    movel([0.183357, -1.188644, -2.683075, -0.840670, 1.570796, 1.754154],accel_mss,speed_ms,0,blend_radius_m)
    movel([0.183318, -1.188232, -2.683266, -0.840892, 1.570796, 1.754114],accel_mss,speed_ms,0,blend_radius_m)
    movel([0.183016, -1.187801, -2.683465, -0.841123, 1.570796, 1.753812],accel_mss,speed_ms,0,blend_radius_m)
    movel([0.182567, -1.187331, -2.683682, -0.841376, 1.570796, 1.753364],accel_mss,speed_ms,0,blend_radius_m)
    movel([0.183152, -1.186492, -2.684069, -0.841828, 1.570796, 1.753948],accel_mss,speed_ms,0,blend_radius_m)
    movel([0.183941, -1.185475, -2.684537, -0.842376, 1.570796, 1.754737],accel_mss,speed_ms,0,blend_radius_m)
    movel([0.184909, -1.184431, -2.685017, -0.842941, 1.570796, 1.755705],accel_mss,speed_ms,0,blend_radius_m)
    movel([0.185946, -1.183470, -2.685457, -0.843461, 1.570796, 1.756743],accel_mss,speed_ms,0,blend_radius_m)
    movel([0.186948, -1.182701, -2.685809, -0.843879, 1.570796, 1.757744],accel_mss,speed_ms,0,blend_radius_m)
    movel([0.187725, -1.182215, -2.686031, -0.844143, 1.570796, 1.758522],accel_mss,speed_ms,0,blend_radius_m)
    movel([0.189510, -1.181449, -2.686380, -0.844559, 1.570796, 1.760306],accel_mss,speed_ms,0,blend_radius_m)
    movel([0.191283, -1.180865, -2.686647, -0.844878, 1.570796, 1.762079],accel_mss,speed_ms,0,blend_radius_m)
    movel([0.194335, -1.179783, -2.687138, -0.845468, 1.570796, 1.765131],accel_mss,speed_ms,0,blend_radius_m)
    movel([0.194860, -1.179431, -2.687298, -0.845660, 1.570796, 1.765656],accel_mss,speed_ms,0,blend_radius_m)
    movel([0.195107, -1.179039, -2.687476, -0.845874, 1.570796, 1.765903],accel_mss,speed_ms,0,blend_radius_m)
    movel([0.194973, -1.178763, -2.687601, -0.846025, 1.570796, 1.765769],accel_mss,speed_ms,0,blend_radius_m)
    movel([0.194450, -1.178756, -2.687604, -0.846029, 1.570796, 1.765246],accel_mss,speed_ms,0,blend_radius_m)
    movel([0.193355, -1.179040, -2.687475, -0.845874, 1.570796, 1.764151],accel_mss,speed_ms,0,blend_radius_m)
    movel([0.188730, -1.180627, -2.686755, -0.845007, 1.570796, 1.759526],accel_mss,speed_ms,0,blend_radius_m)
    movel([0.187737, -1.181042, -2.686566, -0.844781, 1.570796, 1.758533],accel_mss,speed_ms,0,blend_radius_m)
    movel([0.185925, -1.182231, -2.686024, -0.844134, 1.570796, 1.756721],accel_mss,speed_ms,0,blend_radius_m)
    movel([0.184712, -1.183244, -2.685561, -0.843584, 1.570796, 1.755509],accel_mss,speed_ms,0,blend_radius_m)
    movel([0.183607, -1.184345, -2.685056, -0.842987, 1.570796, 1.754403],accel_mss,speed_ms,0,blend_radius_m)
    movel([0.182652, -1.185493, -2.684529, -0.842367, 1.570796, 1.753449],accel_mss,speed_ms,0,blend_radius_m)
    movel([0.181882, -1.186645, -2.683999, -0.841745, 1.570796, 1.752679],accel_mss,speed_ms,0,blend_radius_m)
    movel([0.181412, -1.187532, -2.683589, -0.841268, 1.570796, 1.752208],accel_mss,speed_ms,0,blend_radius_m)
    movel([0.181236, -1.188120, -2.683317, -0.840952, 1.570796, 1.752032],accel_mss,speed_ms,0,blend_radius_m)
    movel([0.181309, -1.188513, -2.683135, -0.840741, 1.570796, 1.752106],accel_mss,speed_ms,0,blend_radius_m)
    movel([0.182133, -1.189002, -2.682909, -0.840478, 1.570796, 1.752929],accel_mss,speed_ms,0,blend_radius_m)
    movel([0.181364, -1.190142, -2.682379, -0.839868, 1.570796, 1.752161],accel_mss,speed_ms,0,blend_radius_m)
    movel([0.180621, -1.191525, -2.681735, -0.839129, 1.570796, 1.751417],accel_mss,speed_ms,0,blend_radius_m)
    movel([0.180458, -1.192089, -2.681472, -0.838828, 1.570796, 1.751254],accel_mss,speed_ms,0,blend_radius_m)
    movel([0.180578, -1.193029, -2.681033, -0.838328, 1.570796, 1.751374],accel_mss,speed_ms,0,blend_radius_m)
    movel([0.180851, -1.193345, -2.680885, -0.838160, 1.570796, 1.751647],accel_mss,speed_ms,0,blend_radius_m)
    movel([0.181819, -1.193755, -2.680692, -0.837942, 1.570796, 1.752615],accel_mss,speed_ms,0,blend_radius_m)
    movel([0.182308, -1.193800, -2.680671, -0.837918, 1.570796, 1.753104],accel_mss,speed_ms,0,blend_radius_m)
    movel([0.188084, -1.193535, -2.680795, -0.838058, 1.570796, 1.758880],accel_mss,speed_ms,0,blend_radius_m)
    movel([0.188322, -1.193692, -2.680722, -0.837975, 1.570796, 1.759118],accel_mss,speed_ms,0,blend_radius_m)
    movel([0.188151, -1.193926, -2.680612, -0.837851, 1.570796, 1.758948],accel_mss,speed_ms,0,blend_radius_m)
    movel([0.185986, -1.194616, -2.680288, -0.837485, 1.570796, 1.756782],accel_mss,speed_ms,0,blend_radius_m)
    movel([0.179630, -1.197004, -2.679163, -0.836222, 1.570796, 1.750426],accel_mss,speed_ms,0,blend_radius_m)
    movel([0.176831, -1.197828, -2.678774, -0.835788, 1.570796, 1.747627],accel_mss,speed_ms,0,blend_radius_m)
    movel([0.174272, -1.198330, -2.678536, -0.835523, 1.570796, 1.745068],accel_mss,speed_ms,0,blend_radius_m)
    movel([0.172010, -1.198496, -2.678457, -0.835436, 1.570796, 1.742806],accel_mss,speed_ms,0,blend_radius_m)
    movel([0.170796, -1.198363, -2.678520, -0.835506, 1.570796, 1.741592],accel_mss,speed_ms,0,blend_radius_m)
    movel([0.170175, -1.197936, -2.678722, -0.835731, 1.570796, 1.740972],accel_mss,speed_ms,0,blend_radius_m)
    movel([0.170106, -1.197645, -2.678860, -0.835884, 1.570796, 1.740903],accel_mss,speed_ms,0,blend_radius_m)
    movel([0.170192, -1.197281, -2.679032, -0.836076, 1.570796, 1.740989],accel_mss,speed_ms,0,blend_radius_m)
    movel([0.171081, -1.196153, -2.679565, -0.836671, 1.570796, 1.741877],accel_mss,speed_ms,0,blend_radius_m)
    movel([0.171201, -1.195957, -2.679657, -0.836775, 1.570796, 1.741997],accel_mss,speed_ms,0,blend_radius_m)
    movel([0.171099, -1.195476, -2.679884, -0.837029, 1.570796, 1.741896],accel_mss,speed_ms,0,blend_radius_m)
    movel([0.170976, -1.195295, -2.679969, -0.837125, 1.570796, 1.741772],accel_mss,speed_ms,0,blend_radius_m)
    movel([0.170326, -1.195000, -2.680108, -0.837281, 1.570796, 1.741123],accel_mss,speed_ms,0,blend_radius_m)
    movel([0.169806, -1.194777, -2.680213, -0.837399, 1.570796, 1.740602],accel_mss,speed_ms,0,blend_radius_m)
    movel([0.169725, -1.194532, -2.680327, -0.837529, 1.570796, 1.740521],accel_mss,speed_ms,0,blend_radius_m)
    movel([0.169784, -1.194220, -2.680474, -0.837695, 1.570796, 1.740581],accel_mss,speed_ms,0,blend_radius_m)
    movel([0.170346, -1.193265, -2.680922, -0.838202, 1.570796, 1.741143],accel_mss,speed_ms,0,blend_radius_m)
    movel([0.171551, -1.191871, -2.681574, -0.838944, 1.570796, 1.742347],accel_mss,speed_ms,0,blend_radius_m)
    movel([0.173401, -1.190152, -2.682375, -0.839862, 1.570796, 1.744197],accel_mss,speed_ms,0,blend_radius_m)
    movel([0.175623, -1.188559, -2.683114, -0.840716, 1.570796, 1.746419],accel_mss,speed_ms,0,blend_radius_m)
    movel([0.177833, -1.187338, -2.683679, -0.841372, 1.570796, 1.748630],accel_mss,speed_ms,0,blend_radius_m)
    movel([0.178746, -1.186974, -2.683847, -0.841568, 1.570796, 1.749542],accel_mss,speed_ms,0,blend_radius_m)
    movel([0.180052, -1.186660, -2.683992, -0.841737, 1.570796, 1.750848],accel_mss,speed_ms,0,blend_radius_m)
    movel([0.180327, -1.186549, -2.684043, -0.841797, 1.570796, 1.751123],accel_mss,speed_ms,0,blend_radius_m)
    movel([0.180720, -1.186157, -2.684224, -0.842008, 1.570796, 1.751516],accel_mss,speed_ms,0,blend_radius_m)
    movel([0.180901, -1.185757, -2.684408, -0.842224, 1.570796, 1.751698],accel_mss,speed_ms,0,blend_radius_m)
    movel([0.180851, -1.185515, -2.684519, -0.842355, 1.570796, 1.751647],accel_mss,speed_ms,0,blend_radius_m)
    movel([0.180544, -1.185423, -2.684562, -0.842405, 1.570796, 1.751341],accel_mss,speed_ms,0,blend_radius_m)
    movel([0.179921, -1.185486, -2.684533, -0.842371, 1.570796, 1.750718],accel_mss,speed_ms,0,blend_radius_m)
    movel([0.178586, -1.185838, -2.684371, -0.842181, 1.570796, 1.749382],accel_mss,speed_ms,0,blend_radius_m)
    movel([0.177208, -1.186449, -2.684089, -0.841851, 1.570796, 1.748004],accel_mss,speed_ms,0,blend_radius_m)
    movel([0.175555, -1.187413, -2.683644, -0.841332, 1.570796, 1.746352],accel_mss,speed_ms,0,blend_radius_m)
    movel([0.173939, -1.188522, -2.683131, -0.840736, 1.570796, 1.744736],accel_mss,speed_ms,0,blend_radius_m)
    movel([0.172391, -1.189757, -2.682558, -0.840074, 1.570796, 1.743187],accel_mss,speed_ms,0,blend_radius_m)
    movel([0.170920, -1.191108, -2.681930, -0.839352, 1.570796, 1.741716],accel_mss,speed_ms,0,blend_radius_m)
    movel([0.169840, -1.192310, -2.681369, -0.838710, 1.570796, 1.740637],accel_mss,speed_ms,0,blend_radius_m)
    movel([0.168953, -1.193603, -2.680764, -0.838022, 1.570796, 1.739749],accel_mss,speed_ms,0,blend_radius_m)
    movel([0.168565, -1.194208, -2.680480, -0.837701, 1.570796, 1.739361],accel_mss,speed_ms,0,blend_radius_m)
    movel([0.167841, -1.194873, -2.680167, -0.837348, 1.570796, 1.738638],accel_mss,speed_ms,0,blend_radius_m)
    movel([0.167132, -1.195268, -2.679981, -0.837139, 1.570796, 1.737928],accel_mss,speed_ms,0,blend_radius_m)
    movel([0.164862, -1.196685, -2.679314, -0.836390, 1.570796, 1.735658],accel_mss,speed_ms,0,blend_radius_m)
    movel([0.162528, -1.198602, -2.678407, -0.835380, 1.570796, 1.733324],accel_mss,speed_ms,0,blend_radius_m)
    movel([0.160445, -1.200728, -2.677396, -0.834265, 1.570796, 1.731242],accel_mss,speed_ms,0,blend_radius_m)
    movel([0.159641, -1.201726, -2.676920, -0.833743, 1.570796, 1.730437],accel_mss,speed_ms,0,blend_radius_m)
    movel([0.158201, -1.203864, -2.675896, -0.832628, 1.570796, 1.728998],accel_mss,speed_ms,0,blend_radius_m)
    movel([0.158043, -1.203914, -2.675872, -0.832602, 1.570796, 1.728839],accel_mss,speed_ms,0,blend_radius_m)
    movel([0.157841, -1.203774, -2.675940, -0.832675, 1.570796, 1.728637],accel_mss,speed_ms,0,blend_radius_m)
    movel([0.157600, -1.203660, -2.675994, -0.832735, 1.570796, 1.728397],accel_mss,speed_ms,0,blend_radius_m)
    movel([0.157314, -1.203744, -2.675954, -0.832691, 1.570796, 1.728111],accel_mss,speed_ms,0,blend_radius_m)
    movel([0.156829, -1.204106, -2.675780, -0.832503, 1.570796, 1.727625],accel_mss,speed_ms,0,blend_radius_m)
    movel([0.153276, -1.207330, -2.674226, -0.830833, 1.570796, 1.724072],accel_mss,speed_ms,0,blend_radius_m)
    movel([0.151027, -1.209704, -2.673074, -0.829610, 1.570796, 1.721823],accel_mss,speed_ms,0,blend_radius_m)
    movel([0.148903, -1.212185, -2.671864, -0.828340, 1.570796, 1.719700],accel_mss,speed_ms,0,blend_radius_m)
    movel([0.147125, -1.214534, -2.670712, -0.827143, 1.570796, 1.717921],accel_mss,speed_ms,0,blend_radius_m)
    movel([0.146009, -1.216173, -2.669904, -0.826312, 1.570796, 1.716805],accel_mss,speed_ms,0,blend_radius_m)
    movel([0.145534, -1.217059, -2.669466, -0.825864, 1.570796, 1.716330],accel_mss,speed_ms,0,blend_radius_m)
    movel([0.145529, -1.217471, -2.669262, -0.825656, 1.570796, 1.716326],accel_mss,speed_ms,0,blend_radius_m)
    movel([0.145867, -1.217578, -2.669209, -0.825602, 1.570796, 1.716664],accel_mss,speed_ms,0,blend_radius_m)
    movel([0.146124, -1.217471, -2.669262, -0.825656, 1.570796, 1.716921],accel_mss,speed_ms,0,blend_radius_m)
    movel([0.146381, -1.217258, -2.669368, -0.825763, 1.570796, 1.717177],accel_mss,speed_ms,0,blend_radius_m)
    movel([0.148924, -1.213700, -2.671122, -0.827568, 1.570796, 1.719721],accel_mss,speed_ms,0,blend_radius_m)
    movel([0.151184, -1.210948, -2.672468, -0.828972, 1.570796, 1.721980],accel_mss,speed_ms,0,blend_radius_m)
    movel([0.153647, -1.208297, -2.673758, -0.830334, 1.570796, 1.724443],accel_mss,speed_ms,0,blend_radius_m)
    movel([0.156117, -1.205971, -2.674882, -0.831535, 1.570796, 1.726914],accel_mss,speed_ms,0,blend_radius_m)
    movel([0.157615, -1.204719, -2.675486, -0.832184, 1.570796, 1.728411],accel_mss,speed_ms,0,blend_radius_m)
    movel([0.157396, -1.205607, -2.675058, -0.831724, 1.570796, 1.728192],accel_mss,speed_ms,0,blend_radius_m)
    movel([0.157289, -1.205968, -2.674884, -0.831537, 1.570796, 1.728085],accel_mss,speed_ms,0,blend_radius_m)
    movel([0.157248, -1.206792, -2.674486, -0.831110, 1.570796, 1.728045],accel_mss,speed_ms,0,blend_radius_m)
    movel([0.157510, -1.207083, -2.674346, -0.830960, 1.570796, 1.728307],accel_mss,speed_ms,0,blend_radius_m)
    movel([0.158082, -1.207177, -2.674300, -0.830912, 1.570796, 1.728878],accel_mss,speed_ms,0,blend_radius_m)
    movel([0.159104, -1.207089, -2.674343, -0.830957, 1.570796, 1.729901],accel_mss,speed_ms,0,blend_radius_m)
    movel([0.161055, -1.206656, -2.674552, -0.831181, 1.570796, 1.731852],accel_mss,speed_ms,0,blend_radius_m)
    movel([0.161633, -1.206359, -2.674695, -0.831334, 1.570796, 1.732429],accel_mss,speed_ms,0,blend_radius_m)
    movel([0.161996, -1.205991, -2.674873, -0.831525, 1.570796, 1.732793],accel_mss,speed_ms,0,blend_radius_m)
    movel([0.162127, -1.205617, -2.675053, -0.831718, 1.570796, 1.732924],accel_mss,speed_ms,0,blend_radius_m)
    movel([0.161992, -1.205417, -2.675150, -0.831822, 1.570796, 1.732788],accel_mss,speed_ms,0,blend_radius_m)
    movel([0.161506, -1.205409, -2.675154, -0.831826, 1.570796, 1.732303],accel_mss,speed_ms,0,blend_radius_m)
    movel([0.159027, -1.205918, -2.674908, -0.831563, 1.570796, 1.729824],accel_mss,speed_ms,0,blend_radius_m)
    movel([0.158633, -1.205765, -2.674982, -0.831642, 1.570796, 1.729429],accel_mss,speed_ms,0,blend_radius_m)
    movel([0.158690, -1.205254, -2.675228, -0.831907, 1.570796, 1.729487],accel_mss,speed_ms,0,blend_radius_m)
    movel([0.159555, -1.203686, -2.675982, -0.832721, 1.570796, 1.730351],accel_mss,speed_ms,0,blend_radius_m)
    movel([0.161064, -1.201525, -2.677016, -0.833848, 1.570796, 1.731861],accel_mss,speed_ms,0,blend_radius_m)
    movel([0.163073, -1.199370, -2.678042, -0.834977, 1.570796, 1.733869],accel_mss,speed_ms,0,blend_radius_m)
    movel([0.165272, -1.197525, -2.678917, -0.835947, 1.570796, 1.736068],accel_mss,speed_ms,0,blend_radius_m)
    movel([0.166291, -1.196848, -2.679237, -0.836304, 1.570796, 1.737087],accel_mss,speed_ms,0,blend_radius_m)
    movel([0.167890, -1.196069, -2.679604, -0.836715, 1.570796, 1.738686],accel_mss,speed_ms,0,blend_radius_m)
    movel([0.168251, -1.195979, -2.679647, -0.836763, 1.570796, 1.739048],accel_mss,speed_ms,0,blend_radius_m)
    movel([0.168882, -1.196151, -2.679566, -0.836672, 1.570796, 1.739679],accel_mss,speed_ms,0,blend_radius_m)
    movel([0.169124, -1.196310, -2.679491, -0.836588, 1.570796, 1.739920],accel_mss,speed_ms,0,blend_radius_m)
    movel([0.169263, -1.196631, -2.679339, -0.836418, 1.570796, 1.740059],accel_mss,speed_ms,0,blend_radius_m)
    movel([0.169187, -1.196810, -2.679255, -0.836324, 1.570796, 1.739984],accel_mss,speed_ms,0,blend_radius_m)
    movel([0.168789, -1.197977, -2.678703, -0.835709, 1.570796, 1.739586],accel_mss,speed_ms,0,blend_radius_m)
    movel([0.168749, -1.198411, -2.678497, -0.835481, 1.570796, 1.739546],accel_mss,speed_ms,0,blend_radius_m)
    movel([0.168985, -1.199003, -2.678217, -0.835170, 1.570796, 1.739781],accel_mss,speed_ms,0,blend_radius_m)
    movel([0.169337, -1.199309, -2.678071, -0.835009, 1.570796, 1.740134],accel_mss,speed_ms,0,blend_radius_m)
    movel([0.170273, -1.199713, -2.677879, -0.834797, 1.570796, 1.741070],accel_mss,speed_ms,0,blend_radius_m)
    movel([0.170932, -1.199776, -2.677850, -0.834764, 1.570796, 1.741729],accel_mss,speed_ms,0,blend_radius_m)
    movel([0.173806, -1.199710, -2.677881, -0.834798, 1.570796, 1.744603],accel_mss,speed_ms,0,blend_radius_m)
    movel([0.169997, -1.201753, -2.676907, -0.833729, 1.570796, 1.740793],accel_mss,speed_ms,0,blend_radius_m)
    movel([0.164056, -1.205160, -2.675273, -0.831955, 1.570796, 1.734852],accel_mss,speed_ms,0,blend_radius_m)
    movel([0.158222, -1.208931, -2.673450, -0.830008, 1.570796, 1.729018],accel_mss,speed_ms,0,blend_radius_m)
    movel([0.155609, -1.210782, -2.672549, -0.829057, 1.570796, 1.726406],accel_mss,speed_ms,0,blend_radius_m)
    movel([0.153043, -1.212728, -2.671598, -0.828063, 1.570796, 1.723839],accel_mss,speed_ms,0,blend_radius_m)
    movel([0.148093, -1.216872, -2.669559, -0.825958, 1.570796, 1.718889],accel_mss,speed_ms,0,blend_radius_m)
    movel([0.145657, -1.219114, -2.668447, -0.824828, 1.570796, 1.716453],accel_mss,speed_ms,0,blend_radius_m)
    movel([0.141026, -1.223786, -2.666112, -0.822491, 1.570796, 1.711822],accel_mss,speed_ms,0,blend_radius_m)
    movel([0.138839, -1.226205, -2.664893, -0.821290, 1.570796, 1.709635],accel_mss,speed_ms,0,blend_radius_m)
    movel([0.134113, -1.231833, -2.662032, -0.818524, 1.570796, 1.704910],accel_mss,speed_ms,0,blend_radius_m)
    movel([0.129720, -1.237546, -2.659090, -0.815754, 1.570796, 1.700516],accel_mss,speed_ms,0,blend_radius_m)
    movel([0.127006, -1.241371, -2.657098, -0.813920, 1.570796, 1.697802],accel_mss,speed_ms,0,blend_radius_m)
    movel([0.124468, -1.245218, -2.655078, -0.812093, 1.570796, 1.695265],accel_mss,speed_ms,0,blend_radius_m)
    movel([0.122226, -1.248912, -2.653121, -0.810355, 1.570796, 1.693023],accel_mss,speed_ms,0,blend_radius_m)
    movel([0.120184, -1.252606, -2.651149, -0.808634, 1.570796, 1.690981],accel_mss,speed_ms,0,blend_radius_m)
    movel([0.118156, -1.256650, -2.648970, -0.806769, 1.570796, 1.688952],accel_mss,speed_ms,0,blend_radius_m)
    movel([0.116335, -1.260667, -2.646787, -0.804935, 1.570796, 1.687131],accel_mss,speed_ms,0,blend_radius_m)
    movel([0.114295, -1.265566, -2.644097, -0.802726, 1.570796, 1.685091],accel_mss,speed_ms,0,blend_radius_m)
    movel([0.112409, -1.270417, -2.641405, -0.800567, 1.570796, 1.683205],accel_mss,speed_ms,0,blend_radius_m)
    movel([0.110443, -1.275872, -2.638343, -0.798175, 1.570796, 1.681240],accel_mss,speed_ms,0,blend_radius_m)
    movel([0.109095, -1.280175, -2.635901, -0.796313, 1.570796, 1.679892],accel_mss,speed_ms,0,blend_radius_m)
    movel([0.108198, -1.283839, -2.633803, -0.794747, 1.570796, 1.678994],accel_mss,speed_ms,0,blend_radius_m)
    movel([0.107629, -1.287288, -2.631813, -0.793288, 1.570796, 1.678425],accel_mss,speed_ms,0,blend_radius_m)
    movel([0.107418, -1.289676, -2.630427, -0.792286, 1.570796, 1.678214],accel_mss,speed_ms,0,blend_radius_m)
    movel([0.107364, -1.291997, -2.629072, -0.791320, 1.570796, 1.678161],accel_mss,speed_ms,0,blend_radius_m)
    movel([0.107481, -1.294116, -2.627829, -0.790444, 1.570796, 1.678278],accel_mss,speed_ms,0,blend_radius_m)
    movel([0.107776, -1.296142, -2.626636, -0.789612, 1.570796, 1.678573],accel_mss,speed_ms,0,blend_radius_m)
    movel([0.108341, -1.298654, -2.625148, -0.788587, 1.570796, 1.679137],accel_mss,speed_ms,0,blend_radius_m)
    movel([0.109047, -1.301076, -2.623707, -0.787607, 1.570796, 1.679843],accel_mss,speed_ms,0,blend_radius_m)
    movel([0.111736, -1.308914, -2.618988, -0.784486, 1.570796, 1.682533],accel_mss,speed_ms,0,blend_radius_m)
    movel([0.113063, -1.312631, -2.616723, -0.783035, 1.570796, 1.683860],accel_mss,speed_ms,0,blend_radius_m)
    movel([0.112154, -1.313491, -2.616196, -0.782702, 1.570796, 1.682950],accel_mss,speed_ms,0,blend_radius_m)
    movel([0.110554, -1.315098, -2.615210, -0.782082, 1.570796, 1.681350],accel_mss,speed_ms,0,blend_radius_m)
    movel([0.105604, -1.320526, -2.611850, -0.780012, 1.570796, 1.676400],accel_mss,speed_ms,0,blend_radius_m)
    movel([0.103992, -1.322440, -2.610657, -0.779292, 1.570796, 1.674788],accel_mss,speed_ms,0,blend_radius_m)
    movel([0.101936, -1.325101, -2.608989, -0.778299, 1.570796, 1.672733],accel_mss,speed_ms,0,blend_radius_m)
    movel([0.100022, -1.327790, -2.607294, -0.777305, 1.570796, 1.670818],accel_mss,speed_ms,0,blend_radius_m)
    movel([0.098207, -1.330560, -2.605538, -0.776291, 1.570796, 1.669003],accel_mss,speed_ms,0,blend_radius_m)
    movel([0.096539, -1.333341, -2.603764, -0.775284, 1.570796, 1.667335],accel_mss,speed_ms,0,blend_radius_m)
    movel([0.095051, -1.336061, -2.602020, -0.774309, 1.570796, 1.665848],accel_mss,speed_ms,0,blend_radius_m)
    movel([0.093714, -1.338778, -2.600266, -0.773345, 1.570796, 1.664510],accel_mss,speed_ms,0,blend_radius_m)
    movel([0.092625, -1.341300, -2.598630, -0.772459, 1.570796, 1.663421],accel_mss,speed_ms,0,blend_radius_m)
    movel([0.091710, -1.343801, -2.596999, -0.771589, 1.570796, 1.662507],accel_mss,speed_ms,0,blend_radius_m)
    movel([0.090931, -1.346349, -2.595328, -0.770712, 1.570796, 1.661727],accel_mss,speed_ms,0,blend_radius_m)
    movel([0.090290, -1.348864, -2.593671, -0.769855, 1.570796, 1.661086],accel_mss,speed_ms,0,blend_radius_m)
    movel([0.089357, -1.353982, -2.590270, -0.768137, 1.570796, 1.660153],accel_mss,speed_ms,0,blend_radius_m)
    movel([0.089065, -1.356593, -2.588520, -0.767275, 1.570796, 1.659861],accel_mss,speed_ms,0,blend_radius_m)
    movel([0.088856, -1.361787, -2.585013, -0.765589, 1.570796, 1.659653],accel_mss,speed_ms,0,blend_radius_m)
    movel([0.088925, -1.364369, -2.583255, -0.764764, 1.570796, 1.659721],accel_mss,speed_ms,0,blend_radius_m)
    movel([0.089318, -1.368741, -2.580258, -0.763390, 1.570796, 1.660114],accel_mss,speed_ms,0,blend_radius_m)
    movel([0.090062, -1.372927, -2.577362, -0.762100, 1.570796, 1.660858],accel_mss,speed_ms,0,blend_radius_m)
    movel([0.091178, -1.377118, -2.574438, -0.760833, 1.570796, 1.661974],accel_mss,speed_ms,0,blend_radius_m)
    movel([0.092594, -1.381119, -2.571623, -0.759647, 1.570796, 1.663390],accel_mss,speed_ms,0,blend_radius_m)
    movel([0.094363, -1.385075, -2.568817, -0.758497, 1.570796, 1.665160],accel_mss,speed_ms,0,blend_radius_m)
    movel([0.096417, -1.388825, -2.566136, -0.757428, 1.570796, 1.667214],accel_mss,speed_ms,0,blend_radius_m)
    movel([0.098800, -1.392482, -2.563503, -0.756405, 1.570796, 1.669596],accel_mss,speed_ms,0,blend_radius_m)
    movel([0.101432, -1.395933, -2.560999, -0.755457, 1.570796, 1.672228],accel_mss,speed_ms,0,blend_radius_m)
    movel([0.103048, -1.397724, -2.559693, -0.754972, 1.570796, 1.673844],accel_mss,speed_ms,0,blend_radius_m)
    movel([0.104830, -1.399364, -2.558493, -0.754532, 1.570796, 1.675626],accel_mss,speed_ms,0,blend_radius_m)
    movel([0.106498, -1.400557, -2.557618, -0.754215, 1.570796, 1.677295],accel_mss,speed_ms,0,blend_radius_m)
    movel([0.108382, -1.401515, -2.556913, -0.753961, 1.570796, 1.679178],accel_mss,speed_ms,0,blend_radius_m)
    movel([0.110318, -1.402168, -2.556432, -0.753789, 1.570796, 1.681114],accel_mss,speed_ms,0,blend_radius_m)
    movel([0.112427, -1.402562, -2.556141, -0.753686, 1.570796, 1.683223],accel_mss,speed_ms,0,blend_radius_m)
    movel([0.114808, -1.402728, -2.556019, -0.753642, 1.570796, 1.685604],accel_mss,speed_ms,0,blend_radius_m)
    movel([0.117295, -1.402659, -2.556070, -0.753660, 1.570796, 1.688091],accel_mss,speed_ms,0,blend_radius_m)
    movel([0.119116, -1.402423, -2.556244, -0.753722, 1.570796, 1.689913],accel_mss,speed_ms,0,blend_radius_m)
    movel([0.121505, -1.401921, -2.556614, -0.753854, 1.570796, 1.692302],accel_mss,speed_ms,0,blend_radius_m)
    movel([0.123903, -1.401300, -2.557071, -0.754018, 1.570796, 1.694699],accel_mss,speed_ms,0,blend_radius_m)
    movel([0.125742, -1.400674, -2.557532, -0.754184, 1.570796, 1.696539],accel_mss,speed_ms,0,blend_radius_m)
    movel([0.129029, -1.399183, -2.558625, -0.754580, 1.570796, 1.699825],accel_mss,speed_ms,0,blend_radius_m)
    movel([0.130586, -1.398328, -2.559251, -0.754809, 1.570796, 1.701382],accel_mss,speed_ms,0,blend_radius_m)
    movel([0.132111, -1.397384, -2.559941, -0.755064, 1.570796, 1.702908],accel_mss,speed_ms,0,blend_radius_m)
    movel([0.133568, -1.396370, -2.560681, -0.755338, 1.570796, 1.704364],accel_mss,speed_ms,0,blend_radius_m)
    movel([0.134973, -1.395280, -2.561474, -0.755635, 1.570796, 1.705769],accel_mss,speed_ms,0,blend_radius_m)
    movel([0.136322, -1.394110, -2.562324, -0.755955, 1.570796, 1.707118],accel_mss,speed_ms,0,blend_radius_m)
    movel([0.137604, -1.392877, -2.563216, -0.756295, 1.570796, 1.708400],accel_mss,speed_ms,0,blend_radius_m)
    movel([0.139420, -1.390830, -2.564695, -0.756864, 1.570796, 1.710217],accel_mss,speed_ms,0,blend_radius_m)
    movel([0.140117, -1.389881, -2.565378, -0.757130, 1.570796, 1.710913],accel_mss,speed_ms,0,blend_radius_m)
    movel([0.140711, -1.388907, -2.566077, -0.757405, 1.570796, 1.711508],accel_mss,speed_ms,0,blend_radius_m)
    movel([0.141155, -1.387998, -2.566729, -0.757662, 1.570796, 1.711951],accel_mss,speed_ms,0,blend_radius_m)
    movel([0.141480, -1.387090, -2.567379, -0.757920, 1.570796, 1.712276],accel_mss,speed_ms,0,blend_radius_m)
    movel([0.141680, -1.386204, -2.568012, -0.758173, 1.570796, 1.712477],accel_mss,speed_ms,0,blend_radius_m)
    movel([0.141752, -1.385350, -2.568621, -0.758418, 1.570796, 1.712549],accel_mss,speed_ms,0,blend_radius_m)
    movel([0.141579, -1.384188, -2.569448, -0.758753, 1.570796, 1.712375],accel_mss,speed_ms,0,blend_radius_m)
    movel([0.141052, -1.383273, -2.570098, -0.759018, 1.570796, 1.711849],accel_mss,speed_ms,0,blend_radius_m)
    movel([0.140042, -1.382449, -2.570682, -0.759258, 1.570796, 1.710838],accel_mss,speed_ms,0,blend_radius_m)
    movel([0.138322, -1.381549, -2.571319, -0.759521, 1.570796, 1.709118],accel_mss,speed_ms,0,blend_radius_m)
    movel([0.135744, -1.380110, -2.572335, -0.759944, 1.570796, 1.706541],accel_mss,speed_ms,0,blend_radius_m)
    movel([0.130444, -1.376520, -2.574857, -0.761012, 1.570796, 1.701240],accel_mss,speed_ms,0,blend_radius_m)
    movel([0.125164, -1.372833, -2.577428, -0.762129, 1.570796, 1.695960],accel_mss,speed_ms,0,blend_radius_m)
    movel([0.122027, -1.370380, -2.579127, -0.762882, 1.570796, 1.692823],accel_mss,speed_ms,0,blend_radius_m)
    movel([0.119338, -1.367897, -2.580839, -0.763653, 1.570796, 1.690134],accel_mss,speed_ms,0,blend_radius_m)
    movel([0.117149, -1.365481, -2.582496, -0.764412, 1.570796, 1.687945],accel_mss,speed_ms,0,blend_radius_m)
    movel([0.115330, -1.362974, -2.584206, -0.765209, 1.570796, 1.686126],accel_mss,speed_ms,0,blend_radius_m)
    movel([0.113763, -1.360220, -2.586075, -0.766094, 1.570796, 1.684560],accel_mss,speed_ms,0,blend_radius_m)
    movel([0.112264, -1.356613, -2.588508, -0.767269, 1.570796, 1.683061],accel_mss,speed_ms,0,blend_radius_m)
    movel([0.111758, -1.354856, -2.589685, -0.767848, 1.570796, 1.682554],accel_mss,speed_ms,0,blend_radius_m)
    movel([0.111393, -1.353018, -2.590913, -0.768458, 1.570796, 1.682190],accel_mss,speed_ms,0,blend_radius_m)
    movel([0.111182, -1.351138, -2.592164, -0.769087, 1.570796, 1.681978],accel_mss,speed_ms,0,blend_radius_m)
    movel([0.111120, -1.349189, -2.593456, -0.769745, 1.570796, 1.681917],accel_mss,speed_ms,0,blend_radius_m)
    movel([0.111200, -1.347063, -2.594858, -0.770467, 1.570796, 1.681997],accel_mss,speed_ms,0,blend_radius_m)
    movel([0.111417, -1.344885, -2.596289, -0.771215, 1.570796, 1.682214],accel_mss,speed_ms,0,blend_radius_m)
    movel([0.112119, -1.340910, -2.598884, -0.772595, 1.570796, 1.682915],accel_mss,speed_ms,0,blend_radius_m)
    movel([0.112599, -1.339021, -2.600109, -0.773259, 1.570796, 1.683395],accel_mss,speed_ms,0,blend_radius_m)
    movel([0.113189, -1.337110, -2.601344, -0.773935, 1.570796, 1.683985],accel_mss,speed_ms,0,blend_radius_m)
    movel([0.114704, -1.333261, -2.603815, -0.775313, 1.570796, 1.685501],accel_mss,speed_ms,0,blend_radius_m)
    movel([0.116745, -1.329144, -2.606437, -0.776808, 1.570796, 1.687541],accel_mss,speed_ms,0,blend_radius_m)
    movel([0.119880, -1.323906, -2.609739, -0.778744, 1.570796, 1.690677],accel_mss,speed_ms,0,blend_radius_m)
    movel([0.120321, -1.323329, -2.610101, -0.778960, 1.570796, 1.691117],accel_mss,speed_ms,0,blend_radius_m)
    movel([0.120558, -1.323269, -2.610138, -0.778982, 1.570796, 1.691354],accel_mss,speed_ms,0,blend_radius_m)
    movel([0.121259, -1.324012, -2.609673, -0.778705, 1.570796, 1.692056],accel_mss,speed_ms,0,blend_radius_m)
    movel([0.124898, -1.328474, -2.606861, -0.777054, 1.570796, 1.695694],accel_mss,speed_ms,0,blend_radius_m)
    movel([0.128998, -1.333445, -2.603698, -0.775246, 1.570796, 1.699794],accel_mss,speed_ms,0,blend_radius_m)
    movel([0.132146, -1.336702, -2.601607, -0.774080, 1.570796, 1.702943],accel_mss,speed_ms,0,blend_radius_m)
    movel([0.135997, -1.339924, -2.599524, -0.772941, 1.570796, 1.706793],accel_mss,speed_ms,0,blend_radius_m)
    movel([0.142877, -1.345098, -2.596150, -0.771141, 1.570796, 1.713674],accel_mss,speed_ms,0,blend_radius_m)
    movel([0.146737, -1.347989, -2.594248, -0.770152, 1.570796, 1.717533],accel_mss,speed_ms,0,blend_radius_m)
    movel([0.145430, -1.350508, -2.592582, -0.769299, 1.570796, 1.716226],accel_mss,speed_ms,0,blend_radius_m)
    movel([0.144148, -1.353044, -2.590896, -0.768449, 1.570796, 1.714944],accel_mss,speed_ms,0,blend_radius_m)
    movel([0.143499, -1.354516, -2.589912, -0.767960, 1.570796, 1.714295],accel_mss,speed_ms,0,blend_radius_m)
    movel([0.143109, -1.355763, -2.589078, -0.767548, 1.570796, 1.713905],accel_mss,speed_ms,0,blend_radius_m)
    movel([0.142789, -1.357342, -2.588017, -0.767030, 1.570796, 1.713585],accel_mss,speed_ms,0,blend_radius_m)
    movel([0.142603, -1.358764, -2.587059, -0.766566, 1.570796, 1.713399],accel_mss,speed_ms,0,blend_radius_m)
    movel([0.142636, -1.359633, -2.586473, -0.766284, 1.570796, 1.713432],accel_mss,speed_ms,0,blend_radius_m)
    movel([0.142888, -1.360224, -2.586073, -0.766092, 1.570796, 1.713684],accel_mss,speed_ms,0,blend_radius_m)
    movel([0.143400, -1.360709, -2.585744, -0.765936, 1.570796, 1.714197],accel_mss,speed_ms,0,blend_radius_m)
    movel([0.144238, -1.360996, -2.585550, -0.765843, 1.570796, 1.715035],accel_mss,speed_ms,0,blend_radius_m)
    movel([0.145422, -1.360988, -2.585555, -0.765846, 1.570796, 1.716218],accel_mss,speed_ms,0,blend_radius_m)
    movel([0.146844, -1.360690, -2.585757, -0.765942, 1.570796, 1.717640],accel_mss,speed_ms,0,blend_radius_m)
    movel([0.148392, -1.360123, -2.586141, -0.766125, 1.570796, 1.719189],accel_mss,speed_ms,0,blend_radius_m)
    movel([0.150333, -1.359097, -2.586834, -0.766457, 1.570796, 1.721129],accel_mss,speed_ms,0,blend_radius_m)
    movel([0.152645, -1.357534, -2.587888, -0.766967, 1.570796, 1.723442],accel_mss,speed_ms,0,blend_radius_m)
    movel([0.154989, -1.355690, -2.589126, -0.767572, 1.570796, 1.725785],accel_mss,speed_ms,0,blend_radius_m)
    movel([0.157035, -1.353806, -2.590387, -0.768196, 1.570796, 1.727831],accel_mss,speed_ms,0,blend_radius_m)
    movel([0.157857, -1.352980, -2.590939, -0.768471, 1.570796, 1.728653],accel_mss,speed_ms,0,blend_radius_m)
    movel([0.160075, -1.353110, -2.590851, -0.768427, 1.570796, 1.730871],accel_mss,speed_ms,0,blend_radius_m)
    movel([0.163680, -1.353196, -2.590794, -0.768399, 1.570796, 1.734476],accel_mss,speed_ms,0,blend_radius_m)
    movel([0.166554, -1.352939, -2.590966, -0.768484, 1.570796, 1.737350],accel_mss,speed_ms,0,blend_radius_m)
    movel([0.167816, -1.352675, -2.591142, -0.768572, 1.570796, 1.738612],accel_mss,speed_ms,0,blend_radius_m)
    movel([0.169098, -1.352297, -2.591393, -0.768699, 1.570796, 1.739894],accel_mss,speed_ms,0,blend_radius_m)
    movel([0.170370, -1.351809, -2.591718, -0.768862, 1.570796, 1.741166],accel_mss,speed_ms,0,blend_radius_m)
    movel([0.171634, -1.351213, -2.592114, -0.769062, 1.570796, 1.742430],accel_mss,speed_ms,0,blend_radius_m)
    movel([0.172833, -1.350504, -2.592584, -0.769300, 1.570796, 1.743629],accel_mss,speed_ms,0,blend_radius_m)
    movel([0.174191, -1.349527, -2.593232, -0.769630, 1.570796, 1.744987],accel_mss,speed_ms,0,blend_radius_m)
    movel([0.175450, -1.348490, -2.593917, -0.769981, 1.570796, 1.746247],accel_mss,speed_ms,0,blend_radius_m)
    movel([0.176314, -1.347609, -2.594499, -0.770281, 1.570796, 1.747111],accel_mss,speed_ms,0,blend_radius_m)
    movel([0.177079, -1.346528, -2.595211, -0.770651, 1.570796, 1.747876],accel_mss,speed_ms,0,blend_radius_m)
    movel([0.177589, -1.345410, -2.595945, -0.771034, 1.570796, 1.748385],accel_mss,speed_ms,0,blend_radius_m)
    movel([0.177789, -1.344366, -2.596630, -0.771394, 1.570796, 1.748585],accel_mss,speed_ms,0,blend_radius_m)
    movel([0.177666, -1.343435, -2.597238, -0.771716, 1.570796, 1.748462],accel_mss,speed_ms,0,blend_radius_m)
    movel([0.177157, -1.342384, -2.597924, -0.772081, 1.570796, 1.747953],accel_mss,speed_ms,0,blend_radius_m)
    movel([0.176397, -1.341524, -2.598484, -0.772381, 1.570796, 1.747193],accel_mss,speed_ms,0,blend_radius_m)
    movel([0.175032, -1.340441, -2.599188, -0.772760, 1.570796, 1.745828],accel_mss,speed_ms,0,blend_radius_m)
    movel([0.171836, -1.338404, -2.600508, -0.773477, 1.570796, 1.742632],accel_mss,speed_ms,0,blend_radius_m)
    movel([0.174790, -1.334338, -2.603126, -0.774925, 1.570796, 1.745587],accel_mss,speed_ms,0,blend_radius_m)
    movel([0.180012, -1.327030, -2.607774, -0.777585, 1.570796, 1.750808],accel_mss,speed_ms,0,blend_radius_m)
    movel([0.182142, -1.323855, -2.609771, -0.778763, 1.570796, 1.752938],accel_mss,speed_ms,0,blend_radius_m)
    movel([0.184172, -1.320639, -2.611780, -0.779970, 1.570796, 1.754969],accel_mss,speed_ms,0,blend_radius_m)
    movel([0.185962, -1.317607, -2.613661, -0.781120, 1.570796, 1.756758],accel_mss,speed_ms,0,blend_radius_m)
    movel([0.187641, -1.314548, -2.615547, -0.782293, 1.570796, 1.758437],accel_mss,speed_ms,0,blend_radius_m)
    movel([0.190775, -1.308160, -2.619446, -0.784783, 1.570796, 1.761571],accel_mss,speed_ms,0,blend_radius_m)
    movel([0.192358, -1.304508, -2.621651, -0.786231, 1.570796, 1.763154],accel_mss,speed_ms,0,blend_radius_m)
    movel([0.193800, -1.300842, -2.623846, -0.787701, 1.570796, 1.764596],accel_mss,speed_ms,0,blend_radius_m)
    movel([0.194919, -1.297593, -2.625777, -0.789018, 1.570796, 1.765715],accel_mss,speed_ms,0,blend_radius_m)
    movel([0.195843, -1.294355, -2.627689, -0.790345, 1.570796, 1.766640],accel_mss,speed_ms,0,blend_radius_m)
    movel([0.196460, -1.291558, -2.629329, -0.791502, 1.570796, 1.767256],accel_mss,speed_ms,0,blend_radius_m)
    movel([0.196871, -1.288804, -2.630934, -0.792651, 1.570796, 1.767667],accel_mss,speed_ms,0,blend_radius_m)
    movel([0.196992, -1.286510, -2.632263, -0.793615, 1.570796, 1.767788],accel_mss,speed_ms,0,blend_radius_m)
    movel([0.196820, -1.284332, -2.633520, -0.794537, 1.570796, 1.767616],accel_mss,speed_ms,0,blend_radius_m)
    movel([0.196320, -1.282324, -2.634672, -0.795392, 1.570796, 1.767116],accel_mss,speed_ms,0,blend_radius_m)
    movel([0.195454, -1.280548, -2.635688, -0.796153, 1.570796, 1.766251],accel_mss,speed_ms,0,blend_radius_m)
    movel([0.194188, -1.278914, -2.636618, -0.796856, 1.570796, 1.764984],accel_mss,speed_ms,0,blend_radius_m)
    movel([0.192628, -1.277541, -2.637398, -0.797450, 1.570796, 1.763425],accel_mss,speed_ms,0,blend_radius_m)
    movel([0.190710, -1.276389, -2.638050, -0.797950, 1.570796, 1.761506],accel_mss,speed_ms,0,blend_radius_m)
    movel([0.188541, -1.275536, -2.638532, -0.798321, 1.570796, 1.759338],accel_mss,speed_ms,0,blend_radius_m)
    movel([0.186099, -1.274972, -2.638850, -0.798567, 1.570796, 1.756895],accel_mss,speed_ms,0,blend_radius_m)
    movel([0.183474, -1.274713, -2.638996, -0.798680, 1.570796, 1.754270],accel_mss,speed_ms,0,blend_radius_m)
    movel([0.180252, -1.274725, -2.638990, -0.798675, 1.570796, 1.751048],accel_mss,speed_ms,0,blend_radius_m)
    movel([0.177190, -1.275011, -2.638829, -0.798550, 1.570796, 1.747986],accel_mss,speed_ms,0,blend_radius_m)
    movel([0.173859, -1.275627, -2.638481, -0.798281, 1.570796, 1.744655],accel_mss,speed_ms,0,blend_radius_m)
    movel([0.169793, -1.276654, -2.637900, -0.797834, 1.570796, 1.740589],accel_mss,speed_ms,0,blend_radius_m)
    movel([0.165350, -1.277999, -2.637138, -0.797251, 1.570796, 1.736146],accel_mss,speed_ms,0,blend_radius_m)
    movel([0.160886, -1.279579, -2.636240, -0.796570, 1.570796, 1.731682],accel_mss,speed_ms,0,blend_radius_m)
    movel([0.156345, -1.281410, -2.635196, -0.795783, 1.570796, 1.727141],accel_mss,speed_ms,0,blend_radius_m)
    movel([0.151813, -1.283453, -2.634025, -0.794911, 1.570796, 1.722609],accel_mss,speed_ms,0,blend_radius_m)
    movel([0.147442, -1.285633, -2.632770, -0.793986, 1.570796, 1.718238],accel_mss,speed_ms,0,blend_radius_m)
    movel([0.143115, -1.288005, -2.631398, -0.792986, 1.570796, 1.713911],accel_mss,speed_ms,0,blend_radius_m)
    movel([0.139175, -1.290387, -2.630013, -0.791990, 1.570796, 1.709972],accel_mss,speed_ms,0,blend_radius_m)
    movel([0.133132, -1.294452, -2.627632, -0.790305, 1.570796, 1.703928],accel_mss,speed_ms,0,blend_radius_m)
    movel([0.132834, -1.294379, -2.627675, -0.790335, 1.570796, 1.703630],accel_mss,speed_ms,0,blend_radius_m)
    movel([0.132761, -1.294194, -2.627784, -0.790412, 1.570796, 1.703557],accel_mss,speed_ms,0,blend_radius_m)
    movel([0.132196, -1.290062, -2.630202, -0.792125, 1.570796, 1.702992],accel_mss,speed_ms,0,blend_radius_m)
    movel([0.131569, -1.284958, -2.633160, -0.794272, 1.570796, 1.702365],accel_mss,speed_ms,0,blend_radius_m)
    movel([0.130827, -1.278139, -2.637059, -0.797191, 1.570796, 1.701623],accel_mss,speed_ms,0,blend_radius_m)
    movel([0.130777, -1.273982, -2.639408, -0.798999, 1.570796, 1.701574],accel_mss,speed_ms,0,blend_radius_m)
    movel([0.131068, -1.269664, -2.641824, -0.800900, 1.570796, 1.701864],accel_mss,speed_ms,0,blend_radius_m)
    movel([0.131694, -1.265511, -2.644127, -0.802750, 1.570796, 1.702490],accel_mss,speed_ms,0,blend_radius_m)
    movel([0.132719, -1.261220, -2.646484, -0.804684, 1.570796, 1.703516],accel_mss,speed_ms,0,blend_radius_m)
    movel([0.134029, -1.257227, -2.648658, -0.806504, 1.570796, 1.704825],accel_mss,speed_ms,0,blend_radius_m)
    movel([0.135723, -1.253166, -2.650848, -0.808375, 1.570796, 1.706519],accel_mss,speed_ms,0,blend_radius_m)
    movel([0.137642, -1.249500, -2.652809, -0.810080, 1.570796, 1.708438],accel_mss,speed_ms,0,blend_radius_m)
    movel([0.139992, -1.245872, -2.654733, -0.811784, 1.570796, 1.710788],accel_mss,speed_ms,0,blend_radius_m)
    movel([0.142133, -1.243089, -2.656198, -0.813102, 1.570796, 1.712929],accel_mss,speed_ms,0,blend_radius_m)
    movel([0.144399, -1.240580, -2.657511, -0.814298, 1.570796, 1.715195],accel_mss,speed_ms,0,blend_radius_m)
    movel([0.147135, -1.237990, -2.658859, -0.815540, 1.570796, 1.717931],accel_mss,speed_ms,0,blend_radius_m)
    movel([0.150755, -1.234924, -2.660445, -0.817020, 1.570796, 1.721551],accel_mss,speed_ms,0,blend_radius_m)
    movel([0.153491, -1.232768, -2.661553, -0.818068, 1.570796, 1.724288],accel_mss,speed_ms,0,blend_radius_m)
    movel([0.156293, -1.230710, -2.662606, -0.819073, 1.570796, 1.727089],accel_mss,speed_ms,0,blend_radius_m)
    movel([0.159028, -1.228848, -2.663554, -0.819987, 1.570796, 1.729824],accel_mss,speed_ms,0,blend_radius_m)
    movel([0.161810, -1.227112, -2.664435, -0.820842, 1.570796, 1.732606],accel_mss,speed_ms,0,blend_radius_m)
    movel([0.164554, -1.225553, -2.665223, -0.821613, 1.570796, 1.735350],accel_mss,speed_ms,0,blend_radius_m)
    movel([0.167321, -1.224134, -2.665937, -0.822318, 1.570796, 1.738117],accel_mss,speed_ms,0,blend_radius_m)
    movel([0.170084, -1.222871, -2.666571, -0.822946, 1.570796, 1.740881],accel_mss,speed_ms,0,blend_radius_m)
    movel([0.172843, -1.221765, -2.667125, -0.823499, 1.570796, 1.743639],accel_mss,speed_ms,0,blend_radius_m)
    movel([0.176034, -1.220676, -2.667669, -0.824044, 1.570796, 1.746830],accel_mss,speed_ms,0,blend_radius_m)
    movel([0.179192, -1.219796, -2.668108, -0.824485, 1.570796, 1.749988],accel_mss,speed_ms,0,blend_radius_m)
    movel([0.182296, -1.219132, -2.668438, -0.824819, 1.570796, 1.753092],accel_mss,speed_ms,0,blend_radius_m)
    movel([0.185332, -1.218686, -2.668660, -0.825044, 1.570796, 1.756129],accel_mss,speed_ms,0,blend_radius_m)
    movel([0.188617, -1.218408, -2.668798, -0.825183, 1.570796, 1.759413],accel_mss,speed_ms,0,blend_radius_m)
    movel([0.191824, -1.218313, -2.668845, -0.825231, 1.570796, 1.762620],accel_mss,speed_ms,0,blend_radius_m)
    movel([0.194941, -1.218406, -2.668798, -0.825184, 1.570796, 1.765737],accel_mss,speed_ms,0,blend_radius_m)
    movel([0.197960, -1.218685, -2.668660, -0.825044, 1.570796, 1.768756],accel_mss,speed_ms,0,blend_radius_m)
    movel([0.201114, -1.219176, -2.668416, -0.824797, 1.570796, 1.771910],accel_mss,speed_ms,0,blend_radius_m)
    movel([0.204151, -1.219854, -2.668079, -0.824456, 1.570796, 1.774947],accel_mss,speed_ms,0,blend_radius_m)
    movel([0.207064, -1.220713, -2.667651, -0.824025, 1.570796, 1.777860],accel_mss,speed_ms,0,blend_radius_m)
    movel([0.209845, -1.221752, -2.667132, -0.823505, 1.570796, 1.780641],accel_mss,speed_ms,0,blend_radius_m)
    movel([0.212626, -1.223013, -2.666500, -0.822876, 1.570796, 1.783422],accel_mss,speed_ms,0,blend_radius_m)
    movel([0.215278, -1.224432, -2.665787, -0.822170, 1.570796, 1.786074],accel_mss,speed_ms,0,blend_radius_m)
    movel([0.217790, -1.226005, -2.664994, -0.821389, 1.570796, 1.788586],accel_mss,speed_ms,0,blend_radius_m)
    movel([0.220162, -1.227729, -2.664122, -0.820538, 1.570796, 1.790958],accel_mss,speed_ms,0,blend_radius_m)
    movel([0.223904, -1.231003, -2.662456, -0.818930, 1.570796, 1.794701],accel_mss,speed_ms,0,blend_radius_m)
    movel([0.228006, -1.235315, -2.660243, -0.816831, 1.570796, 1.798802],accel_mss,speed_ms,0,blend_radius_m)
    movel([0.231738, -1.239820, -2.657908, -0.814661, 1.570796, 1.802534],accel_mss,speed_ms,0,blend_radius_m)
    movel([0.234360, -1.243683, -2.655886, -0.812820, 1.570796, 1.805156],accel_mss,speed_ms,0,blend_radius_m)
    movel([0.235086, -1.245032, -2.655176, -0.812181, 1.570796, 1.805882],accel_mss,speed_ms,0,blend_radius_m)
    movel([0.237133, -1.249550, -2.652782, -0.810057, 1.570796, 1.807929],accel_mss,speed_ms,0,blend_radius_m)
    movel([0.238488, -1.252806, -2.651042, -0.808542, 1.570796, 1.809284],accel_mss,speed_ms,0,blend_radius_m)
    movel([0.240687, -1.257549, -2.648484, -0.806357, 1.570796, 1.811483],accel_mss,speed_ms,0,blend_radius_m)
    movel([0.241968, -1.259887, -2.647212, -0.805290, 1.570796, 1.812764],accel_mss,speed_ms,0,blend_radius_m)
    movel([0.245606, -1.265608, -2.644074, -0.802707, 1.570796, 1.816402],accel_mss,speed_ms,0,blend_radius_m)
    movel([0.247931, -1.268862, -2.642271, -0.801256, 1.570796, 1.818727],accel_mss,speed_ms,0,blend_radius_m)
    movel([0.249805, -1.271133, -2.641005, -0.800251, 1.570796, 1.820601],accel_mss,speed_ms,0,blend_radius_m)
    movel([0.251890, -1.273204, -2.639845, -0.799340, 1.570796, 1.822687],accel_mss,speed_ms,0,blend_radius_m)
    movel([0.253739, -1.274658, -2.639027, -0.798704, 1.570796, 1.824536],accel_mss,speed_ms,0,blend_radius_m)
    movel([0.255797, -1.275884, -2.638336, -0.798169, 1.570796, 1.826594],accel_mss,speed_ms,0,blend_radius_m)
    movel([0.257840, -1.276723, -2.637862, -0.797805, 1.570796, 1.828636],accel_mss,speed_ms,0,blend_radius_m)
    movel([0.260101, -1.277256, -2.637560, -0.797573, 1.570796, 1.830897],accel_mss,speed_ms,0,blend_radius_m)
    movel([0.261706, -1.277392, -2.637483, -0.797514, 1.570796, 1.832503],accel_mss,speed_ms,0,blend_radius_m)
    movel([0.262463, -1.277326, -2.637520, -0.797543, 1.570796, 1.833259],accel_mss,speed_ms,0,blend_radius_m)
    movel([0.264624, -1.276924, -2.637748, -0.797717, 1.570796, 1.835421],accel_mss,speed_ms,0,blend_radius_m)
    movel([0.265315, -1.276722, -2.637862, -0.797805, 1.570796, 1.836112],accel_mss,speed_ms,0,blend_radius_m)
    movel([0.266874, -1.275943, -2.638302, -0.798143, 1.570796, 1.837671],accel_mss,speed_ms,0,blend_radius_m)
    movel([0.268546, -1.274823, -2.638935, -0.798632, 1.570796, 1.839342],accel_mss,speed_ms,0,blend_radius_m)
    movel([0.270080, -1.273462, -2.639700, -0.799227, 1.570796, 1.840876],accel_mss,speed_ms,0,blend_radius_m)
    movel([0.271699, -1.271680, -2.640699, -0.800010, 1.570796, 1.842495],accel_mss,speed_ms,0,blend_radius_m)
    movel([0.273137, -1.269798, -2.641750, -0.800841, 1.570796, 1.843933],accel_mss,speed_ms,0,blend_radius_m)
    movel([0.274692, -1.267398, -2.643084, -0.801907, 1.570796, 1.845488],accel_mss,speed_ms,0,blend_radius_m)
    movel([0.276035, -1.264955, -2.644434, -0.803000, 1.570796, 1.846832],accel_mss,speed_ms,0,blend_radius_m)
    movel([0.277470, -1.261933, -2.646094, -0.804361, 1.570796, 1.848266],accel_mss,speed_ms,0,blend_radius_m)
    movel([0.278749, -1.258899, -2.647750, -0.805740, 1.570796, 1.849546],accel_mss,speed_ms,0,blend_radius_m)
    movel([0.279792, -1.256043, -2.649299, -0.807048, 1.570796, 1.850588],accel_mss,speed_ms,0,blend_radius_m)
    movel([0.280937, -1.252440, -2.651238, -0.808711, 1.570796, 1.851733],accel_mss,speed_ms,0,blend_radius_m)
    movel([0.281947, -1.248907, -2.653124, -0.810358, 1.570796, 1.852743],accel_mss,speed_ms,0,blend_radius_m)
    movel([0.282533, -1.246344, -2.654483, -0.811562, 1.570796, 1.853330],accel_mss,speed_ms,0,blend_radius_m)
    movel([0.283197, -1.241983, -2.656778, -0.813628, 1.570796, 1.853993],accel_mss,speed_ms,0,blend_radius_m)
    movel([0.283523, -1.237715, -2.659002, -0.815672, 1.570796, 1.854319],accel_mss,speed_ms,0,blend_radius_m)
    movel([0.283479, -1.233825, -2.661010, -0.817553, 1.570796, 1.854275],accel_mss,speed_ms,0,blend_radius_m)
    movel([0.283043, -1.230109, -2.662913, -0.819368, 1.570796, 1.853839],accel_mss,speed_ms,0,blend_radius_m)
    movel([0.282261, -1.226880, -2.664552, -0.820957, 1.570796, 1.853058],accel_mss,speed_ms,0,blend_radius_m)
    movel([0.281091, -1.223891, -2.666059, -0.822438, 1.570796, 1.851888],accel_mss,speed_ms,0,blend_radius_m)
    movel([0.279622, -1.221464, -2.667276, -0.823649, 1.570796, 1.850419],accel_mss,speed_ms,0,blend_radius_m)
    movel([0.277711, -1.219413, -2.668298, -0.824678, 1.570796, 1.848507],accel_mss,speed_ms,0,blend_radius_m)
    movel([0.277195, -1.218975, -2.668516, -0.824898, 1.570796, 1.847991],accel_mss,speed_ms,0,blend_radius_m)
    movel([0.275411, -1.217730, -2.669134, -0.825525, 1.570796, 1.846207],accel_mss,speed_ms,0,blend_radius_m)
    movel([0.275180, -1.217679, -2.669159, -0.825551, 1.570796, 1.845977],accel_mss,speed_ms,0,blend_radius_m)
    movel([0.274733, -1.217926, -2.669037, -0.825427, 1.570796, 1.845529],accel_mss,speed_ms,0,blend_radius_m)
    movel([0.274454, -1.218317, -2.668843, -0.825229, 1.570796, 1.845250],accel_mss,speed_ms,0,blend_radius_m)
    movel([0.274431, -1.218669, -2.668668, -0.825052, 1.570796, 1.845227],accel_mss,speed_ms,0,blend_radius_m)
    movel([0.274718, -1.219045, -2.668481, -0.824863, 1.570796, 1.845514],accel_mss,speed_ms,0,blend_radius_m)
    movel([0.275443, -1.219562, -2.668224, -0.824603, 1.570796, 1.846240],accel_mss,speed_ms,0,blend_radius_m)
    movel([0.276702, -1.220586, -2.667714, -0.824089, 1.570796, 1.847498],accel_mss,speed_ms,0,blend_radius_m)
    movel([0.278051, -1.222112, -2.666952, -0.823325, 1.570796, 1.848847],accel_mss,speed_ms,0,blend_radius_m)
    movel([0.279279, -1.223850, -2.666080, -0.822459, 1.570796, 1.850075],accel_mss,speed_ms,0,blend_radius_m)
    movel([0.280180, -1.225546, -2.665226, -0.821617, 1.570796, 1.850976],accel_mss,speed_ms,0,blend_radius_m)
    movel([0.281340, -1.228892, -2.663532, -0.819965, 1.570796, 1.852136],accel_mss,speed_ms,0,blend_radius_m)
    movel([0.282009, -1.232528, -2.661676, -0.818185, 1.570796, 1.852805],accel_mss,speed_ms,0,blend_radius_m)
    movel([0.282255, -1.236704, -2.659526, -0.816159, 1.570796, 1.853052],accel_mss,speed_ms,0,blend_radius_m)
    movel([0.282085, -1.241042, -2.657270, -0.814077, 1.570796, 1.852881],accel_mss,speed_ms,0,blend_radius_m)
    movel([0.281490, -1.245646, -2.654852, -0.811891, 1.570796, 1.852286],accel_mss,speed_ms,0,blend_radius_m)
    movel([0.280494, -1.250342, -2.652360, -0.809687, 1.570796, 1.851290],accel_mss,speed_ms,0,blend_radius_m)
    movel([0.279125, -1.255008, -2.649857, -0.807524, 1.570796, 1.849921],accel_mss,speed_ms,0,blend_radius_m)
    movel([0.277369, -1.259701, -2.647314, -0.805374, 1.570796, 1.848165],accel_mss,speed_ms,0,blend_radius_m)
    movel([0.275945, -1.262911, -2.645558, -0.803920, 1.570796, 1.846742],accel_mss,speed_ms,0,blend_radius_m)
    movel([0.274346, -1.266100, -2.643802, -0.802487, 1.570796, 1.845142],accel_mss,speed_ms,0,blend_radius_m)
    movel([0.272901, -1.268536, -2.642452, -0.801401, 1.570796, 1.843698],accel_mss,speed_ms,0,blend_radius_m)
    movel([0.271192, -1.270899, -2.641136, -0.800354, 1.570796, 1.841988],accel_mss,speed_ms,0,blend_radius_m)
    movel([0.269657, -1.272613, -2.640177, -0.799600, 1.570796, 1.840454],accel_mss,speed_ms,0,blend_radius_m)
    movel([0.267920, -1.274148, -2.639315, -0.798927, 1.570796, 1.838716],accel_mss,speed_ms,0,blend_radius_m)
    movel([0.266263, -1.275225, -2.638708, -0.798456, 1.570796, 1.837059],accel_mss,speed_ms,0,blend_radius_m)
    movel([0.264550, -1.275919, -2.638316, -0.798154, 1.570796, 1.835346],accel_mss,speed_ms,0,blend_radius_m)
    movel([0.262822, -1.276237, -2.638137, -0.798016, 1.570796, 1.833618],accel_mss,speed_ms,0,blend_radius_m)
    movel([0.261243, -1.276176, -2.638171, -0.798042, 1.570796, 1.832039],accel_mss,speed_ms,0,blend_radius_m)
    movel([0.259284, -1.275734, -2.638420, -0.798234, 1.570796, 1.830080],accel_mss,speed_ms,0,blend_radius_m)
    movel([0.257461, -1.275091, -2.638783, -0.798515, 1.570796, 1.828257],accel_mss,speed_ms,0,blend_radius_m)
    movel([0.255521, -1.274136, -2.639321, -0.798932, 1.570796, 1.826317],accel_mss,speed_ms,0,blend_radius_m)
    movel([0.253750, -1.272983, -2.639969, -0.799437, 1.570796, 1.824546],accel_mss,speed_ms,0,blend_radius_m)
    movel([0.252100, -1.271601, -2.640743, -0.800045, 1.570796, 1.822896],accel_mss,speed_ms,0,blend_radius_m)
    movel([0.250633, -1.270044, -2.641613, -0.800732, 1.570796, 1.821429],accel_mss,speed_ms,0,blend_radius_m)
    movel([0.248866, -1.267775, -2.642875, -0.801739, 1.570796, 1.819662],accel_mss,speed_ms,0,blend_radius_m)
    movel([0.246707, -1.264682, -2.644585, -0.803123, 1.570796, 1.817503],accel_mss,speed_ms,0,blend_radius_m)
    movel([0.244528, -1.261349, -2.646414, -0.804626, 1.570796, 1.815324],accel_mss,speed_ms,0,blend_radius_m)
    movel([0.241778, -1.256610, -2.648992, -0.806787, 1.570796, 1.812574],accel_mss,speed_ms,0,blend_radius_m)
    movel([0.240917, -1.254836, -2.649950, -0.807603, 1.570796, 1.811714],accel_mss,speed_ms,0,blend_radius_m)
    movel([0.237374, -1.246483, -2.654410, -0.811496, 1.570796, 1.808171],accel_mss,speed_ms,0,blend_radius_m)
    movel([0.236132, -1.243930, -2.655756, -0.812703, 1.570796, 1.806928],accel_mss,speed_ms,0,blend_radius_m)
    movel([0.234829, -1.241692, -2.656930, -0.813767, 1.570796, 1.805625],accel_mss,speed_ms,0,blend_radius_m)
    movel([0.233285, -1.239426, -2.658113, -0.814850, 1.570796, 1.804081],accel_mss,speed_ms,0,blend_radius_m)
    movel([0.229219, -1.234383, -2.660723, -0.817283, 1.570796, 1.800015],accel_mss,speed_ms,0,blend_radius_m)
    movel([0.224630, -1.229682, -2.663130, -0.819577, 1.570796, 1.795426],accel_mss,speed_ms,0,blend_radius_m)
    movel([0.219884, -1.225670, -2.665163, -0.821555, 1.570796, 1.790680],accel_mss,speed_ms,0,blend_radius_m)
    movel([0.217693, -1.224121, -2.665944, -0.822324, 1.570796, 1.788489],accel_mss,speed_ms,0,blend_radius_m)
    movel([0.215367, -1.222720, -2.666647, -0.823022, 1.570796, 1.786163],accel_mss,speed_ms,0,blend_radius_m)
    movel([0.210783, -1.220531, -2.667742, -0.824117, 1.570796, 1.781579],accel_mss,speed_ms,0,blend_radius_m)
    movel([0.205819, -1.218826, -2.668590, -0.824973, 1.570796, 1.776615],accel_mss,speed_ms,0,blend_radius_m)
    movel([0.203304, -1.218192, -2.668905, -0.825292, 1.570796, 1.774101],accel_mss,speed_ms,0,blend_radius_m)
    movel([0.198009, -1.217338, -2.669328, -0.825723, 1.570796, 1.768805],accel_mss,speed_ms,0,blend_radius_m)
    movel([0.195242, -1.217116, -2.669438, -0.825835, 1.570796, 1.766038],accel_mss,speed_ms,0,blend_radius_m)
    movel([0.189870, -1.217111, -2.669440, -0.825837, 1.570796, 1.760666],accel_mss,speed_ms,0,blend_radius_m)
    movel([0.187093, -1.217314, -2.669340, -0.825735, 1.570796, 1.757889],accel_mss,speed_ms,0,blend_radius_m)
    movel([0.181639, -1.218108, -2.668947, -0.825335, 1.570796, 1.752435],accel_mss,speed_ms,0,blend_radius_m)
    movel([0.178971, -1.218718, -2.668644, -0.825027, 1.570796, 1.749768],accel_mss,speed_ms,0,blend_radius_m)
    movel([0.176266, -1.219487, -2.668261, -0.824640, 1.570796, 1.747063],accel_mss,speed_ms,0,blend_radius_m)
    movel([0.173538, -1.220410, -2.667802, -0.824177, 1.570796, 1.744334],accel_mss,speed_ms,0,blend_radius_m)
    movel([0.168794, -1.222334, -2.666840, -0.823214, 1.570796, 1.739590],accel_mss,speed_ms,0,blend_radius_m)
    movel([0.164402, -1.224516, -2.665745, -0.822128, 1.570796, 1.735198],accel_mss,speed_ms,0,blend_radius_m)
    movel([0.159990, -1.227152, -2.664414, -0.820822, 1.570796, 1.730786],accel_mss,speed_ms,0,blend_radius_m)
    movel([0.155194, -1.230446, -2.662740, -0.819202, 1.570796, 1.725990],accel_mss,speed_ms,0,blend_radius_m)
    movel([0.149752, -1.234592, -2.660616, -0.817181, 1.570796, 1.720548],accel_mss,speed_ms,0,blend_radius_m)
    movel([0.147516, -1.236448, -2.659658, -0.816283, 1.570796, 1.718312],accel_mss,speed_ms,0,blend_radius_m)
    movel([0.143551, -1.240132, -2.657745, -0.814512, 1.570796, 1.714347],accel_mss,speed_ms,0,blend_radius_m)
    movel([0.141842, -1.241941, -2.656800, -0.813648, 1.570796, 1.712639],accel_mss,speed_ms,0,blend_radius_m)
    movel([0.140419, -1.243615, -2.655922, -0.812852, 1.570796, 1.711215],accel_mss,speed_ms,0,blend_radius_m)
    movel([0.139127, -1.245344, -2.655011, -0.812033, 1.570796, 1.709924],accel_mss,speed_ms,0,blend_radius_m)
    movel([0.136822, -1.248944, -2.653105, -0.810341, 1.570796, 1.707618],accel_mss,speed_ms,0,blend_radius_m)
    movel([0.134905, -1.252572, -2.651167, -0.808650, 1.570796, 1.705701],accel_mss,speed_ms,0,blend_radius_m)
    movel([0.133173, -1.256572, -2.649012, -0.806804, 1.570796, 1.703969],accel_mss,speed_ms,0,blend_radius_m)
    movel([0.131791, -1.260516, -2.646869, -0.805004, 1.570796, 1.702588],accel_mss,speed_ms,0,blend_radius_m)
    movel([0.130683, -1.264649, -2.644603, -0.803137, 1.570796, 1.701479],accel_mss,speed_ms,0,blend_radius_m)
    movel([0.129931, -1.268672, -2.642377, -0.801341, 1.570796, 1.700727],accel_mss,speed_ms,0,blend_radius_m)
    movel([0.129510, -1.272695, -2.640131, -0.799563, 1.570796, 1.700306],accel_mss,speed_ms,0,blend_radius_m)
    movel([0.129423, -1.276569, -2.637949, -0.797872, 1.570796, 1.700220],accel_mss,speed_ms,0,blend_radius_m)
    movel([0.129513, -1.278326, -2.636953, -0.797110, 1.570796, 1.700309],accel_mss,speed_ms,0,blend_radius_m)
    movel([0.129739, -1.280617, -2.635649, -0.796123, 1.570796, 1.700536],accel_mss,speed_ms,0,blend_radius_m)
    movel([0.131624, -1.295491, -2.627020, -0.789878, 1.570796, 1.702420],accel_mss,speed_ms,0,blend_radius_m)
    movel([0.131659, -1.295737, -2.626874, -0.789777, 1.570796, 1.702455],accel_mss,speed_ms,0,blend_radius_m)
    movel([0.131929, -1.296144, -2.626634, -0.789611, 1.570796, 1.702725],accel_mss,speed_ms,0,blend_radius_m)
    movel([0.132136, -1.296082, -2.626671, -0.789636, 1.570796, 1.702932],accel_mss,speed_ms,0,blend_radius_m)
    movel([0.135704, -1.293754, -2.628042, -0.790593, 1.570796, 1.706500],accel_mss,speed_ms,0,blend_radius_m)
    movel([0.139695, -1.291132, -2.629578, -0.791679, 1.570796, 1.710491],accel_mss,speed_ms,0,blend_radius_m)
    movel([0.143759, -1.288685, -2.631003, -0.792701, 1.570796, 1.714556],accel_mss,speed_ms,0,blend_radius_m)
    movel([0.147951, -1.286384, -2.632336, -0.793669, 1.570796, 1.718747],accel_mss,speed_ms,0,blend_radius_m)
    movel([0.152186, -1.284272, -2.633554, -0.794563, 1.570796, 1.722982],accel_mss,speed_ms,0,blend_radius_m)
    movel([0.156510, -1.282331, -2.634669, -0.795390, 1.570796, 1.727306],accel_mss,speed_ms,0,blend_radius_m)
    movel([0.160846, -1.280601, -2.635658, -0.796130, 1.570796, 1.731643],accel_mss,speed_ms,0,blend_radius_m)
    movel([0.165229, -1.279064, -2.636534, -0.796792, 1.570796, 1.736025],accel_mss,speed_ms,0,blend_radius_m)
    movel([0.169589, -1.277748, -2.637281, -0.797360, 1.570796, 1.740386],accel_mss,speed_ms,0,blend_radius_m)
    movel([0.173175, -1.276819, -2.637807, -0.797763, 1.570796, 1.743972],accel_mss,speed_ms,0,blend_radius_m)
    movel([0.175922, -1.276260, -2.638123, -0.798006, 1.570796, 1.746719],accel_mss,speed_ms,0,blend_radius_m)
    movel([0.178401, -1.275953, -2.638297, -0.798139, 1.570796, 1.749197],accel_mss,speed_ms,0,blend_radius_m)
    movel([0.181101, -1.275827, -2.638368, -0.798194, 1.570796, 1.751897],accel_mss,speed_ms,0,blend_radius_m)
    movel([0.184688, -1.276009, -2.638265, -0.798115, 1.570796, 1.755484],accel_mss,speed_ms,0,blend_radius_m)
    movel([0.186262, -1.276261, -2.638123, -0.798005, 1.570796, 1.757058],accel_mss,speed_ms,0,blend_radius_m)
    movel([0.187759, -1.276640, -2.637909, -0.797841, 1.570796, 1.758555],accel_mss,speed_ms,0,blend_radius_m)
    movel([0.190370, -1.277738, -2.637286, -0.797364, 1.570796, 1.761166],accel_mss,speed_ms,0,blend_radius_m)
    movel([0.191529, -1.278467, -2.636873, -0.797049, 1.570796, 1.762325],accel_mss,speed_ms,0,blend_radius_m)
    movel([0.193527, -1.280288, -2.635836, -0.796265, 1.570796, 1.764323],accel_mss,speed_ms,0,blend_radius_m)
    movel([0.194339, -1.281380, -2.635213, -0.795796, 1.570796, 1.765135],accel_mss,speed_ms,0,blend_radius_m)
    movel([0.194949, -1.282510, -2.634566, -0.795313, 1.570796, 1.765745],accel_mss,speed_ms,0,blend_radius_m)
    movel([0.195391, -1.283754, -2.633852, -0.794783, 1.570796, 1.766187],accel_mss,speed_ms,0,blend_radius_m)
    movel([0.195679, -1.285147, -2.633050, -0.794192, 1.570796, 1.766475],accel_mss,speed_ms,0,blend_radius_m)
    movel([0.195796, -1.286625, -2.632197, -0.793567, 1.570796, 1.766592],accel_mss,speed_ms,0,blend_radius_m)
    movel([0.195768, -1.288384, -2.631178, -0.792827, 1.570796, 1.766565],accel_mss,speed_ms,0,blend_radius_m)
    movel([0.195607, -1.290190, -2.630127, -0.792072, 1.570796, 1.766404],accel_mss,speed_ms,0,blend_radius_m)
    movel([0.195246, -1.292424, -2.628822, -0.791143, 1.570796, 1.766042],accel_mss,speed_ms,0,blend_radius_m)
    movel([0.194702, -1.294695, -2.627488, -0.790205, 1.570796, 1.765499],accel_mss,speed_ms,0,blend_radius_m)
    movel([0.193877, -1.297473, -2.625849, -0.789068, 1.570796, 1.764673],accel_mss,speed_ms,0,blend_radius_m)
    movel([0.192934, -1.300255, -2.624196, -0.787938, 1.570796, 1.763731],accel_mss,speed_ms,0,blend_radius_m)
    movel([0.190488, -1.306422, -2.620497, -0.785470, 1.570796, 1.761285],accel_mss,speed_ms,0,blend_radius_m)
    movel([0.187507, -1.312810, -2.616613, -0.782965, 1.570796, 1.758303],accel_mss,speed_ms,0,blend_radius_m)
    movel([0.186222, -1.315278, -2.615099, -0.782013, 1.570796, 1.757019],accel_mss,speed_ms,0,blend_radius_m)
    movel([0.184841, -1.317723, -2.613590, -0.781076, 1.570796, 1.755637],accel_mss,speed_ms,0,blend_radius_m)
    movel([0.181451, -1.323218, -2.610170, -0.779001, 1.570796, 1.752247],accel_mss,speed_ms,0,blend_radius_m)
    movel([0.177413, -1.329206, -2.606398, -0.776786, 1.570796, 1.748209],accel_mss,speed_ms,0,blend_radius_m)
    movel([0.171913, -1.336786, -2.601553, -0.774050, 1.570796, 1.742709],accel_mss,speed_ms,0,blend_radius_m)
    movel([0.171179, -1.337807, -2.600894, -0.773688, 1.570796, 1.741976],accel_mss,speed_ms,0,blend_radius_m)
    movel([0.170493, -1.338849, -2.600220, -0.773320, 1.570796, 1.741289],accel_mss,speed_ms,0,blend_radius_m)
    movel([0.170532, -1.338970, -2.600142, -0.773277, 1.570796, 1.741328],accel_mss,speed_ms,0,blend_radius_m)
    movel([0.173887, -1.341163, -2.598720, -0.772507, 1.570796, 1.744683],accel_mss,speed_ms,0,blend_radius_m)
    movel([0.175094, -1.342094, -2.598113, -0.772182, 1.570796, 1.745891],accel_mss,speed_ms,0,blend_radius_m)
    movel([0.175934, -1.342957, -2.597551, -0.771882, 1.570796, 1.746731],accel_mss,speed_ms,0,blend_radius_m)
    movel([0.176426, -1.343782, -2.597012, -0.771596, 1.570796, 1.747223],accel_mss,speed_ms,0,blend_radius_m)
    movel([0.176661, -1.344543, -2.596513, -0.771333, 1.570796, 1.747457],accel_mss,speed_ms,0,blend_radius_m)
    movel([0.176666, -1.345179, -2.596096, -0.771113, 1.570796, 1.747462],accel_mss,speed_ms,0,blend_radius_m)
    movel([0.176438, -1.345847, -2.595658, -0.770884, 1.570796, 1.747235],accel_mss,speed_ms,0,blend_radius_m)
    movel([0.175936, -1.346706, -2.595093, -0.770589, 1.570796, 1.746733],accel_mss,speed_ms,0,blend_radius_m)
    movel([0.175241, -1.347603, -2.594503, -0.770283, 1.570796, 1.746037],accel_mss,speed_ms,0,blend_radius_m)
    movel([0.174403, -1.348417, -2.593966, -0.770006, 1.570796, 1.745199],accel_mss,speed_ms,0,blend_radius_m)
    movel([0.173329, -1.349252, -2.593414, -0.769723, 1.570796, 1.744125],accel_mss,speed_ms,0,blend_radius_m)
    movel([0.172195, -1.349984, -2.592929, -0.769476, 1.570796, 1.742991],accel_mss,speed_ms,0,blend_radius_m)
    movel([0.170910, -1.350665, -2.592478, -0.769246, 1.570796, 1.741707],accel_mss,speed_ms,0,blend_radius_m)
    movel([0.169609, -1.351220, -2.592109, -0.769059, 1.570796, 1.740406],accel_mss,speed_ms,0,blend_radius_m)
    movel([0.168278, -1.351658, -2.591818, -0.768912, 1.570796, 1.739074],accel_mss,speed_ms,0,blend_radius_m)
    movel([0.166965, -1.351961, -2.591617, -0.768811, 1.570796, 1.737761],accel_mss,speed_ms,0,blend_radius_m)
    movel([0.164150, -1.352243, -2.591429, -0.768717, 1.570796, 1.734946],accel_mss,speed_ms,0,blend_radius_m)
    movel([0.162465, -1.352235, -2.591435, -0.768719, 1.570796, 1.733262],accel_mss,speed_ms,0,blend_radius_m)
    movel([0.157807, -1.352016, -2.591580, -0.768793, 1.570796, 1.728604],accel_mss,speed_ms,0,blend_radius_m)
    movel([0.155730, -1.353873, -2.590343, -0.768174, 1.570796, 1.726526],accel_mss,speed_ms,0,blend_radius_m)
    movel([0.153521, -1.355842, -2.589025, -0.767522, 1.570796, 1.724317],accel_mss,speed_ms,0,blend_radius_m)
    movel([0.151642, -1.357307, -2.588041, -0.767041, 1.570796, 1.722438],accel_mss,speed_ms,0,blend_radius_m)
    movel([0.149865, -1.358441, -2.587277, -0.766671, 1.570796, 1.720661],accel_mss,speed_ms,0,blend_radius_m)
    movel([0.147977, -1.359393, -2.586635, -0.766362, 1.570796, 1.718774],accel_mss,speed_ms,0,blend_radius_m)
    movel([0.146435, -1.359944, -2.586262, -0.766183, 1.570796, 1.717232],accel_mss,speed_ms,0,blend_radius_m)
    movel([0.145811, -1.360066, -2.586180, -0.766143, 1.570796, 1.716608],accel_mss,speed_ms,0,blend_radius_m)
    movel([0.145222, -1.360084, -2.586167, -0.766137, 1.570796, 1.716018],accel_mss,speed_ms,0,blend_radius_m)
    movel([0.144342, -1.359810, -2.586353, -0.766226, 1.570796, 1.715139],accel_mss,speed_ms,0,blend_radius_m)
    movel([0.143778, -1.359145, -2.586802, -0.766442, 1.570796, 1.714574],accel_mss,speed_ms,0,blend_radius_m)
    movel([0.143608, -1.358519, -2.587224, -0.766645, 1.570796, 1.714404],accel_mss,speed_ms,0,blend_radius_m)
    movel([0.143608, -1.357815, -2.587699, -0.766875, 1.570796, 1.714404],accel_mss,speed_ms,0,blend_radius_m)
    movel([0.144045, -1.355840, -2.589026, -0.767523, 1.570796, 1.714842],accel_mss,speed_ms,0,blend_radius_m)
    movel([0.145059, -1.353255, -2.590755, -0.768379, 1.570796, 1.715856],accel_mss,speed_ms,0,blend_radius_m)
    movel([0.147753, -1.347958, -2.594268, -0.770162, 1.570796, 1.718549],accel_mss,speed_ms,0,blend_radius_m)
    movel([0.147837, -1.347601, -2.594504, -0.770284, 1.570796, 1.718633],accel_mss,speed_ms,0,blend_radius_m)
    movel([0.147772, -1.347339, -2.594677, -0.770373, 1.570796, 1.718568],accel_mss,speed_ms,0,blend_radius_m)
    movel([0.147578, -1.347135, -2.594811, -0.770443, 1.570796, 1.718374],accel_mss,speed_ms,0,blend_radius_m)
    movel([0.141584, -1.342526, -2.597832, -0.772031, 1.570796, 1.712380],accel_mss,speed_ms,0,blend_radius_m)
    movel([0.136070, -1.338290, -2.600582, -0.773517, 1.570796, 1.706866],accel_mss,speed_ms,0,blend_radius_m)
    movel([0.132410, -1.335107, -2.602632, -0.774649, 1.570796, 1.703207],accel_mss,speed_ms,0,blend_radius_m)
    movel([0.129229, -1.331723, -2.604797, -0.775869, 1.570796, 1.700026],accel_mss,speed_ms,0,blend_radius_m)
    movel([0.122038, -1.322905, -2.610366, -0.779118, 1.570796, 1.692834],accel_mss,speed_ms,0,blend_radius_m)
    movel([0.120923, -1.321726, -2.611102, -0.779560, 1.570796, 1.691719],accel_mss,speed_ms,0,blend_radius_m)
    movel([0.120585, -1.321711, -2.611112, -0.779566, 1.570796, 1.691381],accel_mss,speed_ms,0,blend_radius_m)
    movel([0.120174, -1.322046, -2.610903, -0.779440, 1.570796, 1.690971],accel_mss,speed_ms,0,blend_radius_m)
    movel([0.119146, -1.323509, -2.609988, -0.778892, 1.570796, 1.689942],accel_mss,speed_ms,0,blend_radius_m)
    movel([0.117984, -1.325279, -2.608877, -0.778233, 1.570796, 1.688780],accel_mss,speed_ms,0,blend_radius_m)
    movel([0.115343, -1.329857, -2.605984, -0.776547, 1.570796, 1.686140],accel_mss,speed_ms,0,blend_radius_m)
    movel([0.114072, -1.332448, -2.604335, -0.775606, 1.570796, 1.684868],accel_mss,speed_ms,0,blend_radius_m)
    movel([0.112965, -1.335032, -2.602681, -0.774677, 1.570796, 1.683761],accel_mss,speed_ms,0,blend_radius_m)
    movel([0.112025, -1.337592, -2.601032, -0.773764, 1.570796, 1.682821],accel_mss,speed_ms,0,blend_radius_m)
    movel([0.111271, -1.340097, -2.599412, -0.772880, 1.570796, 1.682067],accel_mss,speed_ms,0,blend_radius_m)
    movel([0.110690, -1.342564, -2.597807, -0.772018, 1.570796, 1.681486],accel_mss,speed_ms,0,blend_radius_m)
    movel([0.110289, -1.344979, -2.596227, -0.771182, 1.570796, 1.681086],accel_mss,speed_ms,0,blend_radius_m)
    movel([0.110068, -1.347334, -2.594680, -0.770375, 1.570796, 1.680864],accel_mss,speed_ms,0,blend_radius_m)
    movel([0.110019, -1.349669, -2.593138, -0.769582, 1.570796, 1.680815],accel_mss,speed_ms,0,blend_radius_m)
    movel([0.110143, -1.351929, -2.591638, -0.768822, 1.570796, 1.680940],accel_mss,speed_ms,0,blend_radius_m)
    movel([0.110444, -1.354103, -2.590189, -0.768097, 1.570796, 1.681240],accel_mss,speed_ms,0,blend_radius_m)
    movel([0.110915, -1.356188, -2.588793, -0.767408, 1.570796, 1.681711],accel_mss,speed_ms,0,blend_radius_m)
    movel([0.111571, -1.358269, -2.587393, -0.766727, 1.570796, 1.682367],accel_mss,speed_ms,0,blend_radius_m)
    movel([0.112379, -1.360255, -2.586052, -0.766082, 1.570796, 1.683175],accel_mss,speed_ms,0,blend_radius_m)
    movel([0.113330, -1.362142, -2.584772, -0.765475, 1.570796, 1.684127],accel_mss,speed_ms,0,blend_radius_m)
    movel([0.114428, -1.363922, -2.583560, -0.764906, 1.570796, 1.685225],accel_mss,speed_ms,0,blend_radius_m)
    movel([0.116685, -1.366856, -2.581553, -0.763979, 1.570796, 1.687481],accel_mss,speed_ms,0,blend_radius_m)
    movel([0.119376, -1.369631, -2.579644, -0.763114, 1.570796, 1.690172],accel_mss,speed_ms,0,blend_radius_m)
    movel([0.122665, -1.372413, -2.577719, -0.762257, 1.570796, 1.693461],accel_mss,speed_ms,0,blend_radius_m)
    movel([0.126724, -1.375369, -2.575661, -0.761359, 1.570796, 1.697520],accel_mss,speed_ms,0,blend_radius_m)
    movel([0.133959, -1.380248, -2.572238, -0.759903, 1.570796, 1.704755],accel_mss,speed_ms,0,blend_radius_m)
    movel([0.136505, -1.381863, -2.571097, -0.759429, 1.570796, 1.707302],accel_mss,speed_ms,0,blend_radius_m)
    movel([0.139400, -1.383402, -2.570006, -0.758981, 1.570796, 1.710197],accel_mss,speed_ms,0,blend_radius_m)
    movel([0.140149, -1.384001, -2.569581, -0.758807, 1.570796, 1.710945],accel_mss,speed_ms,0,blend_radius_m)
    movel([0.140546, -1.384685, -2.569095, -0.758609, 1.570796, 1.711342],accel_mss,speed_ms,0,blend_radius_m)
    movel([0.140717, -1.385618, -2.568430, -0.758341, 1.570796, 1.711513],accel_mss,speed_ms,0,blend_radius_m)
    movel([0.140659, -1.386481, -2.567815, -0.758094, 1.570796, 1.711455],accel_mss,speed_ms,0,blend_radius_m)
    movel([0.140395, -1.387457, -2.567117, -0.757816, 1.570796, 1.711191],accel_mss,speed_ms,0,blend_radius_m)
    movel([0.139931, -1.388528, -2.566350, -0.757512, 1.570796, 1.710727],accel_mss,speed_ms,0,blend_radius_m)
    movel([0.139276, -1.389673, -2.565528, -0.757189, 1.570796, 1.710073],accel_mss,speed_ms,0,blend_radius_m)
    movel([0.138659, -1.390557, -2.564891, -0.756941, 1.570796, 1.709456],accel_mss,speed_ms,0,blend_radius_m)
    movel([0.137954, -1.391411, -2.564276, -0.756702, 1.570796, 1.708750],accel_mss,speed_ms,0,blend_radius_m)
    movel([0.136057, -1.393344, -2.562879, -0.756166, 1.570796, 1.706853],accel_mss,speed_ms,0,blend_radius_m)
    movel([0.133859, -1.395226, -2.561513, -0.755650, 1.570796, 1.704656],accel_mss,speed_ms,0,blend_radius_m)
    movel([0.131605, -1.396828, -2.560347, -0.755214, 1.570796, 1.702401],accel_mss,speed_ms,0,blend_radius_m)
    movel([0.128928, -1.398374, -2.559218, -0.754797, 1.570796, 1.699725],accel_mss,speed_ms,0,blend_radius_m)
    movel([0.126184, -1.399626, -2.558301, -0.754462, 1.570796, 1.696980],accel_mss,speed_ms,0,blend_radius_m)
    movel([0.123295, -1.400627, -2.557566, -0.754196, 1.570796, 1.694091],accel_mss,speed_ms,0,blend_radius_m)
    movel([0.120435, -1.401326, -2.557052, -0.754011, 1.570796, 1.691232],accel_mss,speed_ms,0,blend_radius_m)
    movel([0.117610, -1.401724, -2.556759, -0.753906, 1.570796, 1.688406],accel_mss,speed_ms,0,blend_radius_m)
    movel([0.114893, -1.401802, -2.556702, -0.753885, 1.570796, 1.685690],accel_mss,speed_ms,0,blend_radius_m)
    movel([0.112383, -1.401562, -2.556878, -0.753949, 1.570796, 1.683180],accel_mss,speed_ms,0,blend_radius_m)
    movel([0.110073, -1.400990, -2.557299, -0.754100, 1.570796, 1.680869],accel_mss,speed_ms,0,blend_radius_m)
    movel([0.108794, -1.400475, -2.557678, -0.754236, 1.570796, 1.679590],accel_mss,speed_ms,0,blend_radius_m)
    movel([0.107395, -1.399730, -2.558225, -0.754435, 1.570796, 1.678191],accel_mss,speed_ms,0,blend_radius_m)
    movel([0.106061, -1.398872, -2.558853, -0.754664, 1.570796, 1.676858],accel_mss,speed_ms,0,blend_radius_m)
    movel([0.104983, -1.398011, -2.559483, -0.754895, 1.570796, 1.675779],accel_mss,speed_ms,0,blend_radius_m)
    movel([0.103065, -1.396095, -2.560881, -0.755413, 1.570796, 1.673861],accel_mss,speed_ms,0,blend_radius_m)
    movel([0.101334, -1.394017, -2.562391, -0.755981, 1.570796, 1.672131],accel_mss,speed_ms,0,blend_radius_m)
    movel([0.099435, -1.391364, -2.564309, -0.756715, 1.570796, 1.670232],accel_mss,speed_ms,0,blend_radius_m)
    movel([0.097667, -1.388603, -2.566295, -0.757490, 1.570796, 1.668463],accel_mss,speed_ms,0,blend_radius_m)
    movel([0.095983, -1.385649, -2.568408, -0.758332, 1.570796, 1.666780],accel_mss,speed_ms,0,blend_radius_m)
    movel([0.094441, -1.382587, -2.570584, -0.759218, 1.570796, 1.665237],accel_mss,speed_ms,0,blend_radius_m)
    movel([0.093210, -1.379726, -2.572606, -0.760057, 1.570796, 1.664007],accel_mss,speed_ms,0,blend_radius_m)
    movel([0.092169, -1.376739, -2.574703, -0.760946, 1.570796, 1.662965],accel_mss,speed_ms,0,blend_radius_m)
    movel([0.091454, -1.374211, -2.576469, -0.761709, 1.570796, 1.662251],accel_mss,speed_ms,0,blend_radius_m)
    movel([0.090862, -1.371609, -2.578277, -0.762504, 1.570796, 1.661659],accel_mss,speed_ms,0,blend_radius_m)
    movel([0.090427, -1.369066, -2.580034, -0.763289, 1.570796, 1.661223],accel_mss,speed_ms,0,blend_radius_m)
    movel([0.090129, -1.366447, -2.581834, -0.764108, 1.570796, 1.660925],accel_mss,speed_ms,0,blend_radius_m)
    movel([0.089974, -1.363758, -2.583673, -0.764959, 1.570796, 1.660771],accel_mss,speed_ms,0,blend_radius_m)
    movel([0.089959, -1.361000, -2.585547, -0.765842, 1.570796, 1.660755],accel_mss,speed_ms,0,blend_radius_m)
    movel([0.090086, -1.358033, -2.587552, -0.766804, 1.570796, 1.660883],accel_mss,speed_ms,0,blend_radius_m)
    movel([0.090345, -1.355007, -2.589584, -0.767798, 1.570796, 1.661141],accel_mss,speed_ms,0,blend_radius_m)
    movel([0.090728, -1.351799, -2.591725, -0.768865, 1.570796, 1.661524],accel_mss,speed_ms,0,blend_radius_m)
    movel([0.091129, -1.349390, -2.593322, -0.769676, 1.570796, 1.661925],accel_mss,speed_ms,0,blend_radius_m)
    movel([0.091658, -1.347147, -2.594803, -0.770439, 1.570796, 1.662454],accel_mss,speed_ms,0,blend_radius_m)
    movel([0.092432, -1.344513, -2.596533, -0.771343, 1.570796, 1.663229],accel_mss,speed_ms,0,blend_radius_m)
    movel([0.093724, -1.340950, -2.598858, -0.772581, 1.570796, 1.664520],accel_mss,speed_ms,0,blend_radius_m)
    movel([0.095352, -1.337351, -2.601188, -0.773850, 1.570796, 1.666148],accel_mss,speed_ms,0,blend_radius_m)
    movel([0.097384, -1.333563, -2.603622, -0.775204, 1.570796, 1.668180],accel_mss,speed_ms,0,blend_radius_m)
    movel([0.099707, -1.329784, -2.606031, -0.776574, 1.570796, 1.670503],accel_mss,speed_ms,0,blend_radius_m)
    movel([0.102356, -1.325970, -2.608442, -0.777977, 1.570796, 1.673152],accel_mss,speed_ms,0,blend_radius_m)
    movel([0.105269, -1.322214, -2.610798, -0.779377, 1.570796, 1.676066],accel_mss,speed_ms,0,blend_radius_m)
    movel([0.108408, -1.318582, -2.613058, -0.780749, 1.570796, 1.679204],accel_mss,speed_ms,0,blend_radius_m)
    movel([0.113516, -1.313266, -2.616334, -0.782789, 1.570796, 1.684312],accel_mss,speed_ms,0,blend_radius_m)
    movel([0.114081, -1.312620, -2.616730, -0.783039, 1.570796, 1.684877],accel_mss,speed_ms,0,blend_radius_m)
    movel([0.114194, -1.312387, -2.616873, -0.783130, 1.570796, 1.684990],accel_mss,speed_ms,0,blend_radius_m)
    movel([0.114179, -1.312160, -2.617011, -0.783218, 1.570796, 1.684975],accel_mss,speed_ms,0,blend_radius_m)
    movel([0.110593, -1.301862, -2.623237, -0.787290, 1.570796, 1.681389],accel_mss,speed_ms,0,blend_radius_m)
    movel([0.109587, -1.298609, -2.625175, -0.788605, 1.570796, 1.680383],accel_mss,speed_ms,0,blend_radius_m)
    movel([0.108992, -1.295942, -2.626753, -0.789693, 1.570796, 1.679788],accel_mss,speed_ms,0,blend_radius_m)
    movel([0.108601, -1.293043, -2.628459, -0.790887, 1.570796, 1.679398],accel_mss,speed_ms,0,blend_radius_m)
    movel([0.108486, -1.290903, -2.629711, -0.791775, 1.570796, 1.679283],accel_mss,speed_ms,0,blend_radius_m)
    movel([0.108546, -1.288683, -2.631004, -0.792702, 1.570796, 1.679342],accel_mss,speed_ms,0,blend_radius_m)
    movel([0.108778, -1.286429, -2.632310, -0.793650, 1.570796, 1.679575],accel_mss,speed_ms,0,blend_radius_m)
    movel([0.109194, -1.284113, -2.633646, -0.794630, 1.570796, 1.679990],accel_mss,speed_ms,0,blend_radius_m)
    movel([0.109867, -1.281336, -2.635238, -0.795815, 1.570796, 1.680663],accel_mss,speed_ms,0,blend_radius_m)
    movel([0.110710, -1.278516, -2.636845, -0.797028, 1.570796, 1.681507],accel_mss,speed_ms,0,blend_radius_m)
    movel([0.113408, -1.270809, -2.641186, -0.800394, 1.570796, 1.684204],accel_mss,speed_ms,0,blend_radius_m)
    movel([0.115448, -1.265539, -2.644112, -0.802738, 1.570796, 1.686245],accel_mss,speed_ms,0,blend_radius_m)
    movel([0.117654, -1.260210, -2.647036, -0.805143, 1.570796, 1.688451],accel_mss,speed_ms,0,blend_radius_m)
    movel([0.119539, -1.256070, -2.649284, -0.807035, 1.570796, 1.690335],accel_mss,speed_ms,0,blend_radius_m)
    movel([0.121673, -1.251904, -2.651525, -0.808960, 1.570796, 1.692470],accel_mss,speed_ms,0,blend_radius_m)
    movel([0.123896, -1.248010, -2.653601, -0.810778, 1.570796, 1.694693],accel_mss,speed_ms,0,blend_radius_m)
    movel([0.126359, -1.244127, -2.655653, -0.812609, 1.570796, 1.697155],accel_mss,speed_ms,0,blend_radius_m)
    movel([0.129431, -1.239659, -2.657991, -0.814738, 1.570796, 1.700227],accel_mss,speed_ms,0,blend_radius_m)
    movel([0.132681, -1.235212, -2.660296, -0.816881, 1.570796, 1.703477],accel_mss,speed_ms,0,blend_radius_m)
    movel([0.136891, -1.229869, -2.663035, -0.819485, 1.570796, 1.707687],accel_mss,speed_ms,0,blend_radius_m)
    movel([0.141096, -1.225036, -2.665483, -0.821870, 1.570796, 1.711892],accel_mss,speed_ms,0,blend_radius_m)
    movel([0.145368, -1.220642, -2.667686, -0.824061, 1.570796, 1.716164],accel_mss,speed_ms,0,blend_radius_m)
    movel([0.149769, -1.216618, -2.669684, -0.826087, 1.570796, 1.720565],accel_mss,speed_ms,0,blend_radius_m)
    movel([0.152739, -1.214159, -2.670896, -0.827334, 1.570796, 1.723535],accel_mss,speed_ms,0,blend_radius_m)
    movel([0.155790, -1.211814, -2.672046, -0.828530, 1.570796, 1.726586],accel_mss,speed_ms,0,blend_radius_m)
    movel([0.158908, -1.209591, -2.673129, -0.829668, 1.570796, 1.729704],accel_mss,speed_ms,0,blend_radius_m)
    movel([0.162082, -1.207505, -2.674142, -0.830743, 1.570796, 1.732878],accel_mss,speed_ms,0,blend_radius_m)
    movel([0.165575, -1.205374, -2.675171, -0.831845, 1.570796, 1.736372],accel_mss,speed_ms,0,blend_radius_m)
    movel([0.169099, -1.203372, -2.676133, -0.832885, 1.570796, 1.739895],accel_mss,speed_ms,0,blend_radius_m)
    movel([0.172646, -1.201503, -2.677026, -0.833859, 1.570796, 1.743442],accel_mss,speed_ms,0,blend_radius_m)
    movel([0.176206, -1.199775, -2.677850, -0.834764, 1.570796, 1.747003],accel_mss,speed_ms,0,blend_radius_m)
    movel([0.179897, -1.198133, -2.678629, -0.835627, 1.570796, 1.750693],accel_mss,speed_ms,0,blend_radius_m)
    movel([0.183583, -1.196643, -2.679334, -0.836412, 1.570796, 1.754379],accel_mss,speed_ms,0,blend_radius_m)
    movel([0.187260, -1.195308, -2.679963, -0.837118, 1.570796, 1.758056],accel_mss,speed_ms,0,blend_radius_m)
    movel([0.190913, -1.194130, -2.680516, -0.837742, 1.570796, 1.761709],accel_mss,speed_ms,0,blend_radius_m)
    movel([0.194487, -1.193133, -2.680984, -0.838272, 1.570796, 1.765283],accel_mss,speed_ms,0,blend_radius_m)
    movel([0.198016, -1.192310, -2.681369, -0.838710, 1.570796, 1.768813],accel_mss,speed_ms,0,blend_radius_m)
    movel([0.201500, -1.191658, -2.681673, -0.839058, 1.570796, 1.772297],accel_mss,speed_ms,0,blend_radius_m)
    movel([0.204925, -1.191179, -2.681896, -0.839313, 1.570796, 1.775721],accel_mss,speed_ms,0,blend_radius_m)
    movel([0.209671, -1.190795, -2.682075, -0.839518, 1.570796, 1.780467],accel_mss,speed_ms,0,blend_radius_m)
    movel([0.214275, -1.190737, -2.682103, -0.839550, 1.570796, 1.785072],accel_mss,speed_ms,0,blend_radius_m)
    movel([0.218718, -1.191011, -2.681975, -0.839403, 1.570796, 1.789514],accel_mss,speed_ms,0,blend_radius_m)
    movel([0.222976, -1.191612, -2.681695, -0.839083, 1.570796, 1.793772],accel_mss,speed_ms,0,blend_radius_m)
    movel([0.226916, -1.192520, -2.681270, -0.838598, 1.570796, 1.797713],accel_mss,speed_ms,0,blend_radius_m)
    movel([0.230642, -1.193741, -2.680699, -0.837949, 1.570796, 1.801438],accel_mss,speed_ms,0,blend_radius_m)
    movel([0.233922, -1.195214, -2.680007, -0.837168, 1.570796, 1.804718],accel_mss,speed_ms,0,blend_radius_m)
    movel([0.236929, -1.197018, -2.679157, -0.836214, 1.570796, 1.807725],accel_mss,speed_ms,0,blend_radius_m)
    movel([0.240458, -1.199814, -2.677831, -0.834744, 1.570796, 1.811255],accel_mss,speed_ms,0,blend_radius_m)
    movel([0.243518, -1.203017, -2.676302, -0.833069, 1.570796, 1.814314],accel_mss,speed_ms,0,blend_radius_m)
    movel([0.246054, -1.206552, -2.674602, -0.831235, 1.570796, 1.816851],accel_mss,speed_ms,0,blend_radius_m)
    movel([0.248020, -1.210340, -2.672765, -0.829284, 1.570796, 1.818817],accel_mss,speed_ms,0,blend_radius_m)
    movel([0.248948, -1.212694, -2.671615, -0.828080, 1.570796, 1.819744],accel_mss,speed_ms,0,blend_radius_m)
    movel([0.250903, -1.218817, -2.668595, -0.824977, 1.570796, 1.821700],accel_mss,speed_ms,0,blend_radius_m)
    movel([0.251673, -1.221759, -2.667128, -0.823502, 1.570796, 1.822469],accel_mss,speed_ms,0,blend_radius_m)
    movel([0.252256, -1.224586, -2.665710, -0.822093, 1.570796, 1.823052],accel_mss,speed_ms,0,blend_radius_m)
    movel([0.252313, -1.225370, -2.665315, -0.821704, 1.570796, 1.823110],accel_mss,speed_ms,0,blend_radius_m)
    movel([0.252119, -1.226392, -2.664799, -0.821198, 1.570796, 1.822915],accel_mss,speed_ms,0,blend_radius_m)
    movel([0.252114, -1.226648, -2.664669, -0.821071, 1.570796, 1.822911],accel_mss,speed_ms,0,blend_radius_m)
    movel([0.252664, -1.227115, -2.664433, -0.820840, 1.570796, 1.823460],accel_mss,speed_ms,0,blend_radius_m)
    movel([0.252892, -1.227914, -2.664028, -0.820447, 1.570796, 1.823688],accel_mss,speed_ms,0,blend_radius_m)
    movel([0.253520, -1.231694, -2.662103, -0.818592, 1.570796, 1.824316],accel_mss,speed_ms,0,blend_radius_m)
    movel([0.254096, -1.235374, -2.660213, -0.816803, 1.570796, 1.824892],accel_mss,speed_ms,0,blend_radius_m)
    movel([0.255273, -1.240979, -2.657303, -0.814107, 1.570796, 1.826070],accel_mss,speed_ms,0,blend_radius_m)
    movel([0.255921, -1.243115, -2.656184, -0.813089, 1.570796, 1.826717],accel_mss,speed_ms,0,blend_radius_m)
    movel([0.256893, -1.245588, -2.654883, -0.811918, 1.570796, 1.827689],accel_mss,speed_ms,0,blend_radius_m)
    movel([0.258056, -1.247911, -2.653653, -0.810825, 1.570796, 1.828852],accel_mss,speed_ms,0,blend_radius_m)
    movel([0.259299, -1.249832, -2.652632, -0.809925, 1.570796, 1.830095],accel_mss,speed_ms,0,blend_radius_m)
    movel([0.260770, -1.251552, -2.651713, -0.809124, 1.570796, 1.831566],accel_mss,speed_ms,0,blend_radius_m)
    movel([0.262149, -1.252766, -2.651063, -0.808560, 1.570796, 1.832945],accel_mss,speed_ms,0,blend_radius_m)
    movel([0.263720, -1.253774, -2.650522, -0.808094, 1.570796, 1.834516],accel_mss,speed_ms,0,blend_radius_m)
    movel([0.265017, -1.254154, -2.650317, -0.807918, 1.570796, 1.835813],accel_mss,speed_ms,0,blend_radius_m)
    movel([0.266576, -1.254061, -2.650367, -0.807961, 1.570796, 1.837372],accel_mss,speed_ms,0,blend_radius_m)
    movel([0.268162, -1.253521, -2.650657, -0.808210, 1.570796, 1.838958],accel_mss,speed_ms,0,blend_radius_m)
    movel([0.268641, -1.253267, -2.650794, -0.808328, 1.570796, 1.839437],accel_mss,speed_ms,0,blend_radius_m)
    movel([0.270173, -1.252133, -2.651402, -0.808854, 1.570796, 1.840969],accel_mss,speed_ms,0,blend_radius_m)
    movel([0.271779, -1.250504, -2.652273, -0.809612, 1.570796, 1.842575],accel_mss,speed_ms,0,blend_radius_m)
    movel([0.273303, -1.248559, -2.653309, -0.810521, 1.570796, 1.844100],accel_mss,speed_ms,0,blend_radius_m)
    movel([0.274592, -1.246469, -2.654417, -0.811503, 1.570796, 1.845389],accel_mss,speed_ms,0,blend_radius_m)
    movel([0.275448, -1.244543, -2.655434, -0.812412, 1.570796, 1.846245],accel_mss,speed_ms,0,blend_radius_m)
    movel([0.276254, -1.241932, -2.656805, -0.813652, 1.570796, 1.847050],accel_mss,speed_ms,0,blend_radius_m)
    movel([0.276891, -1.239150, -2.658257, -0.814983, 1.570796, 1.847687],accel_mss,speed_ms,0,blend_radius_m)
    movel([0.277227, -1.236646, -2.659556, -0.816187, 1.570796, 1.848023],accel_mss,speed_ms,0,blend_radius_m)
    movel([0.277345, -1.234191, -2.660822, -0.817376, 1.570796, 1.848141],accel_mss,speed_ms,0,blend_radius_m)
    movel([0.277297, -1.231803, -2.662047, -0.818539, 1.570796, 1.848093],accel_mss,speed_ms,0,blend_radius_m)
    movel([0.277086, -1.229560, -2.663192, -0.819637, 1.570796, 1.847882],accel_mss,speed_ms,0,blend_radius_m)
    movel([0.276698, -1.227409, -2.664285, -0.820696, 1.570796, 1.847494],accel_mss,speed_ms,0,blend_radius_m)
    movel([0.276147, -1.225413, -2.665293, -0.821683, 1.570796, 1.846943],accel_mss,speed_ms,0,blend_radius_m)
    movel([0.275424, -1.223525, -2.666243, -0.822621, 1.570796, 1.846220],accel_mss,speed_ms,0,blend_radius_m)
    movel([0.274540, -1.221803, -2.667106, -0.823480, 1.570796, 1.845336],accel_mss,speed_ms,0,blend_radius_m)
    movel([0.273482, -1.220215, -2.667899, -0.824275, 1.570796, 1.844278],accel_mss,speed_ms,0,blend_radius_m)
    movel([0.272482, -1.219065, -2.668471, -0.824852, 1.570796, 1.843279],accel_mss,speed_ms,0,blend_radius_m)
    movel([0.272133, -1.218838, -2.668584, -0.824967, 1.570796, 1.842930],accel_mss,speed_ms,0,blend_radius_m)
    movel([0.271831, -1.218816, -2.668595, -0.824978, 1.570796, 1.842627],accel_mss,speed_ms,0,blend_radius_m)
    movel([0.271376, -1.219063, -2.668473, -0.824854, 1.570796, 1.842172],accel_mss,speed_ms,0,blend_radius_m)
    movel([0.271187, -1.219431, -2.668289, -0.824668, 1.570796, 1.841984],accel_mss,speed_ms,0,blend_radius_m)
    movel([0.271361, -1.219988, -2.668012, -0.824389, 1.570796, 1.842158],accel_mss,speed_ms,0,blend_radius_m)
    movel([0.271964, -1.220817, -2.667599, -0.823973, 1.570796, 1.842761],accel_mss,speed_ms,0,blend_radius_m)
    movel([0.273182, -1.222548, -2.666734, -0.823108, 1.570796, 1.843978],accel_mss,speed_ms,0,blend_radius_m)
    movel([0.274184, -1.224447, -2.665780, -0.822162, 1.570796, 1.844980],accel_mss,speed_ms,0,blend_radius_m)
    movel([0.274992, -1.226530, -2.664729, -0.821130, 1.570796, 1.845788],accel_mss,speed_ms,0,blend_radius_m)
    movel([0.275580, -1.228751, -2.663604, -0.820035, 1.570796, 1.846376],accel_mss,speed_ms,0,blend_radius_m)
    movel([0.275960, -1.231114, -2.662400, -0.818876, 1.570796, 1.846756],accel_mss,speed_ms,0,blend_radius_m)
    movel([0.276124, -1.233583, -2.661135, -0.817671, 1.570796, 1.846920],accel_mss,speed_ms,0,blend_radius_m)
    movel([0.276071, -1.236144, -2.659815, -0.816430, 1.570796, 1.846867],accel_mss,speed_ms,0,blend_radius_m)
    movel([0.275805, -1.238781, -2.658448, -0.815159, 1.570796, 1.846602],accel_mss,speed_ms,0,blend_radius_m)
    movel([0.275419, -1.240897, -2.657346, -0.814146, 1.570796, 1.846215],accel_mss,speed_ms,0,blend_radius_m)
    movel([0.274837, -1.243056, -2.656215, -0.813117, 1.570796, 1.845633],accel_mss,speed_ms,0,blend_radius_m)
    movel([0.274120, -1.244995, -2.655195, -0.812198, 1.570796, 1.844916],accel_mss,speed_ms,0,blend_radius_m)
    movel([0.273176, -1.246938, -2.654169, -0.811282, 1.570796, 1.843972],accel_mss,speed_ms,0,blend_radius_m)
    movel([0.272189, -1.248540, -2.653319, -0.810530, 1.570796, 1.842985],accel_mss,speed_ms,0,blend_radius_m)
    movel([0.271011, -1.250081, -2.652499, -0.809809, 1.570796, 1.841807],accel_mss,speed_ms,0,blend_radius_m)
    movel([0.269852, -1.251241, -2.651879, -0.809268, 1.570796, 1.840649],accel_mss,speed_ms,0,blend_radius_m)
    movel([0.268535, -1.252186, -2.651374, -0.808829, 1.570796, 1.839332],accel_mss,speed_ms,0,blend_radius_m)
    movel([0.267582, -1.252648, -2.651126, -0.808615, 1.570796, 1.838378],accel_mss,speed_ms,0,blend_radius_m)
    movel([0.266683, -1.252879, -2.651002, -0.808507, 1.570796, 1.837480],accel_mss,speed_ms,0,blend_radius_m)
    movel([0.265766, -1.252881, -2.651001, -0.808507, 1.570796, 1.836563],accel_mss,speed_ms,0,blend_radius_m)
    movel([0.264751, -1.252662, -2.651119, -0.808608, 1.570796, 1.835547],accel_mss,speed_ms,0,blend_radius_m)
    movel([0.263859, -1.252274, -2.651327, -0.808788, 1.570796, 1.834655],accel_mss,speed_ms,0,blend_radius_m)
    movel([0.263122, -1.251705, -2.651631, -0.809052, 1.570796, 1.833919],accel_mss,speed_ms,0,blend_radius_m)
    movel([0.260735, -1.249084, -2.653030, -0.810275, 1.570796, 1.831531],accel_mss,speed_ms,0,blend_radius_m)
    movel([0.258421, -1.246199, -2.654560, -0.811630, 1.570796, 1.829217],accel_mss,speed_ms,0,blend_radius_m)
    movel([0.258350, -1.245788, -2.654777, -0.811824, 1.570796, 1.829146],accel_mss,speed_ms,0,blend_radius_m)
    movel([0.258596, -1.245287, -2.655042, -0.812060, 1.570796, 1.829392],accel_mss,speed_ms,0,blend_radius_m)
    movel([0.258596, -1.244631, -2.655387, -0.812370, 1.570796, 1.829393],accel_mss,speed_ms,0,blend_radius_m)
    movel([0.258518, -1.243848, -2.655800, -0.812742, 1.570796, 1.829314],accel_mss,speed_ms,0,blend_radius_m)
    movel([0.258893, -1.242963, -2.656264, -0.813162, 1.570796, 1.829689],accel_mss,speed_ms,0,blend_radius_m)
    movel([0.259695, -1.242085, -2.656725, -0.813579, 1.570796, 1.830491],accel_mss,speed_ms,0,blend_radius_m)
    movel([0.260821, -1.241329, -2.657120, -0.813940, 1.570796, 1.831618],accel_mss,speed_ms,0,blend_radius_m)
    movel([0.261962, -1.240850, -2.657371, -0.814169, 1.570796, 1.832758],accel_mss,speed_ms,0,blend_radius_m)
    movel([0.263259, -1.240549, -2.657527, -0.814312, 1.570796, 1.834056],accel_mss,speed_ms,0,blend_radius_m)
    movel([0.264431, -1.240462, -2.657573, -0.814354, 1.570796, 1.835227],accel_mss,speed_ms,0,blend_radius_m)
    movel([0.265143, -1.240658, -2.657471, -0.814260, 1.570796, 1.835939],accel_mss,speed_ms,0,blend_radius_m)
    movel([0.265362, -1.240773, -2.657411, -0.814205, 1.570796, 1.836158],accel_mss,speed_ms,0,blend_radius_m)
    movel([0.266050, -1.240887, -2.657351, -0.814151, 1.570796, 1.836847],accel_mss,speed_ms,0,blend_radius_m)
    movel([0.266350, -1.240866, -2.657362, -0.814161, 1.570796, 1.837146],accel_mss,speed_ms,0,blend_radius_m)
    movel([0.266402, -1.240980, -2.657303, -0.814107, 1.570796, 1.837198],accel_mss,speed_ms,0,blend_radius_m)
    movel([0.266237, -1.241186, -2.657195, -0.814008, 1.570796, 1.837033],accel_mss,speed_ms,0,blend_radius_m)
    movel([0.265247, -1.241887, -2.656828, -0.813674, 1.570796, 1.836043],accel_mss,speed_ms,0,blend_radius_m)
    movel([0.264579, -1.242566, -2.656473, -0.813351, 1.570796, 1.835376],accel_mss,speed_ms,0,blend_radius_m)
    movel([0.263427, -1.244142, -2.655645, -0.812602, 1.570796, 1.834224],accel_mss,speed_ms,0,blend_radius_m)
    movel([0.262984, -1.245097, -2.655142, -0.812150, 1.570796, 1.833780],accel_mss,speed_ms,0,blend_radius_m)
    movel([0.262406, -1.247398, -2.653925, -0.811066, 1.570796, 1.833203],accel_mss,speed_ms,0,blend_radius_m)
    movel([0.262377, -1.248322, -2.653435, -0.810632, 1.570796, 1.833173],accel_mss,speed_ms,0,blend_radius_m)
    movel([0.262798, -1.250016, -2.652534, -0.809839, 1.570796, 1.833595],accel_mss,speed_ms,0,blend_radius_m)
    movel([0.263763, -1.251456, -2.651764, -0.809168, 1.570796, 1.834559],accel_mss,speed_ms,0,blend_radius_m)
    movel([0.264797, -1.252084, -2.651429, -0.808877, 1.570796, 1.835593],accel_mss,speed_ms,0,blend_radius_m)
    movel([0.265194, -1.252000, -2.651474, -0.808915, 1.570796, 1.835990],accel_mss,speed_ms,0,blend_radius_m)
    movel([0.265517, -1.251643, -2.651665, -0.809082, 1.570796, 1.836314],accel_mss,speed_ms,0,blend_radius_m)
    movel([0.265537, -1.251456, -2.651764, -0.809168, 1.570796, 1.836334],accel_mss,speed_ms,0,blend_radius_m)
    movel([0.264819, -1.250247, -2.652411, -0.809732, 1.570796, 1.835616],accel_mss,speed_ms,0,blend_radius_m)
    movel([0.264102, -1.249179, -2.652979, -0.810230, 1.570796, 1.834899],accel_mss,speed_ms,0,blend_radius_m)
    movel([0.263717, -1.248165, -2.653518, -0.810705, 1.570796, 1.834513],accel_mss,speed_ms,0,blend_radius_m)
    movel([0.263635, -1.247105, -2.654081, -0.811204, 1.570796, 1.834431],accel_mss,speed_ms,0,blend_radius_m)
    movel([0.263836, -1.245902, -2.654717, -0.811770, 1.570796, 1.834632],accel_mss,speed_ms,0,blend_radius_m)
    movel([0.264366, -1.244503, -2.655455, -0.812431, 1.570796, 1.835162],accel_mss,speed_ms,0,blend_radius_m)
    movel([0.265141, -1.243328, -2.656073, -0.812988, 1.570796, 1.835937],accel_mss,speed_ms,0,blend_radius_m)
    movel([0.266125, -1.242431, -2.656543, -0.813414, 1.570796, 1.836921],accel_mss,speed_ms,0,blend_radius_m)
    movel([0.267647, -1.241694, -2.656929, -0.813766, 1.570796, 1.838444],accel_mss,speed_ms,0,blend_radius_m)
    movel([0.268011, -1.241513, -2.657024, -0.813852, 1.570796, 1.838807],accel_mss,speed_ms,0,blend_radius_m)
    movel([0.268485, -1.241158, -2.657209, -0.814021, 1.570796, 1.839281],accel_mss,speed_ms,0,blend_radius_m)
    movel([0.268713, -1.241026, -2.657278, -0.814084, 1.570796, 1.839509],accel_mss,speed_ms,0,blend_radius_m)
    movel([0.268748, -1.241410, -2.657078, -0.813901, 1.570796, 1.839544],accel_mss,speed_ms,0,blend_radius_m)
    movel([0.269472, -1.242542, -2.656485, -0.813362, 1.570796, 1.840268],accel_mss,speed_ms,0,blend_radius_m)
    movel([0.270218, -1.243593, -2.655933, -0.812862, 1.570796, 1.841015],accel_mss,speed_ms,0,blend_radius_m)
    movel([0.270715, -1.244043, -2.655697, -0.812649, 1.570796, 1.841511],accel_mss,speed_ms,0,blend_radius_m)
    movel([0.271107, -1.244195, -2.655617, -0.812577, 1.570796, 1.841903],accel_mss,speed_ms,0,blend_radius_m)
    movel([0.271501, -1.244167, -2.655632, -0.812590, 1.570796, 1.842297],accel_mss,speed_ms,0,blend_radius_m)
    movel([0.271816, -1.243974, -2.655733, -0.812682, 1.570796, 1.842613],accel_mss,speed_ms,0,blend_radius_m)
    movel([0.272009, -1.243666, -2.655895, -0.812828, 1.570796, 1.842805],accel_mss,speed_ms,0,blend_radius_m)
    movel([0.272002, -1.243499, -2.655983, -0.812907, 1.570796, 1.842799],accel_mss,speed_ms,0,blend_radius_m)
    movel([0.270423, -1.241210, -2.657183, -0.813997, 1.570796, 1.841220],accel_mss,speed_ms,0,blend_radius_m)
    movel([0.269852, -1.240023, -2.657802, -0.814564, 1.570796, 1.840649],accel_mss,speed_ms,0,blend_radius_m)
    movel([0.269473, -1.238726, -2.658477, -0.815186, 1.570796, 1.840269],accel_mss,speed_ms,0,blend_radius_m)
    movel([0.269282, -1.237334, -2.659200, -0.815856, 1.570796, 1.840079],accel_mss,speed_ms,0,blend_radius_m)
    movel([0.269385, -1.234643, -2.660589, -0.817156, 1.570796, 1.840181],accel_mss,speed_ms,0,blend_radius_m)
    movel([0.269553, -1.233087, -2.661389, -0.817912, 1.570796, 1.840349],accel_mss,speed_ms,0,blend_radius_m)
    movel([0.269726, -1.232780, -2.661547, -0.818062, 1.570796, 1.840522],accel_mss,speed_ms,0,blend_radius_m)
    movel([0.271064, -1.233074, -2.661396, -0.817919, 1.570796, 1.841860],accel_mss,speed_ms,0,blend_radius_m)
    movel([0.272118, -1.233330, -2.661265, -0.817794, 1.570796, 1.842915],accel_mss,speed_ms,0,blend_radius_m)
    movel([0.274209, -1.233442, -2.661207, -0.817740, 1.570796, 1.845005],accel_mss,speed_ms,0,blend_radius_m)
    movel([0.274650, -1.233227, -2.661317, -0.817844, 1.570796, 1.845446],accel_mss,speed_ms,0,blend_radius_m)
    movel([0.274831, -1.232962, -2.661453, -0.817973, 1.570796, 1.845627],accel_mss,speed_ms,0,blend_radius_m)
    movel([0.274895, -1.232796, -2.661539, -0.818054, 1.570796, 1.845691],accel_mss,speed_ms,0,blend_radius_m)
    movel([0.274868, -1.232472, -2.661705, -0.818212, 1.570796, 1.845664],accel_mss,speed_ms,0,blend_radius_m)
    movel([0.274650, -1.232351, -2.661767, -0.818271, 1.570796, 1.845446],accel_mss,speed_ms,0,blend_radius_m)
    movel([0.273622, -1.232213, -2.661838, -0.818339, 1.570796, 1.844418],accel_mss,speed_ms,0,blend_radius_m)
    movel([0.272503, -1.232068, -2.661912, -0.818409, 1.570796, 1.843299],accel_mss,speed_ms,0,blend_radius_m)
    movel([0.271457, -1.231749, -2.662075, -0.818565, 1.570796, 1.842253],accel_mss,speed_ms,0,blend_radius_m)
    movel([0.270643, -1.231335, -2.662286, -0.818767, 1.570796, 1.841439],accel_mss,speed_ms,0,blend_radius_m)
    movel([0.270352, -1.230900, -2.662509, -0.818980, 1.570796, 1.841148],accel_mss,speed_ms,0,blend_radius_m)
    movel([0.270297, -1.230746, -2.662588, -0.819056, 1.570796, 1.841094],accel_mss,speed_ms,0,blend_radius_m)
    movel([0.269838, -1.230421, -2.662753, -0.819214, 1.570796, 1.840634],accel_mss,speed_ms,0,blend_radius_m)
    movel([0.269735, -1.230051, -2.662942, -0.819396, 1.570796, 1.840531],accel_mss,speed_ms,0,blend_radius_m)
    movel([0.269575, -1.227075, -2.664454, -0.820861, 1.570796, 1.840372],accel_mss,speed_ms,0,blend_radius_m)
    movel([0.269978, -1.227005, -2.664489, -0.820895, 1.570796, 1.840774],accel_mss,speed_ms,0,blend_radius_m)
    movel([0.270364, -1.227000, -2.664491, -0.820897, 1.570796, 1.841160],accel_mss,speed_ms,0,blend_radius_m)
    movel([0.272607, -1.226884, -2.664550, -0.820955, 1.570796, 1.843404],accel_mss,speed_ms,0,blend_radius_m)
    movel([0.273200, -1.226702, -2.664642, -0.821045, 1.570796, 1.843996],accel_mss,speed_ms,0,blend_radius_m)
    movel([0.273592, -1.226427, -2.664781, -0.821181, 1.570796, 1.844388],accel_mss,speed_ms,0,blend_radius_m)
    movel([0.273858, -1.226019, -2.664987, -0.821382, 1.570796, 1.844654],accel_mss,speed_ms,0,blend_radius_m)
    movel([0.273809, -1.225748, -2.665124, -0.821517, 1.570796, 1.844605],accel_mss,speed_ms,0,blend_radius_m)
    movel([0.273385, -1.225635, -2.665181, -0.821573, 1.570796, 1.844181],accel_mss,speed_ms,0,blend_radius_m)
    movel([0.272519, -1.225697, -2.665150, -0.821542, 1.570796, 1.843315],accel_mss,speed_ms,0,blend_radius_m)
    movel([0.271938, -1.225740, -2.665128, -0.821521, 1.570796, 1.842734],accel_mss,speed_ms,0,blend_radius_m)
    movel([0.270210, -1.225590, -2.665204, -0.821595, 1.570796, 1.841006],accel_mss,speed_ms,0,blend_radius_m)
    movel([0.269603, -1.225372, -2.665314, -0.821703, 1.570796, 1.840399],accel_mss,speed_ms,0,blend_radius_m)
    movel([0.269293, -1.225101, -2.665450, -0.821837, 1.570796, 1.840089],accel_mss,speed_ms,0,blend_radius_m)
    movel([0.269082, -1.224608, -2.665699, -0.822082, 1.570796, 1.839879],accel_mss,speed_ms,0,blend_radius_m)
    movel([0.268295, -1.220623, -2.667696, -0.824070, 1.570796, 1.839091],accel_mss,speed_ms,0,blend_radius_m)
    movel([0.268094, -1.218191, -2.668905, -0.825293, 1.570796, 1.838890],accel_mss,speed_ms,0,blend_radius_m)
    movel([0.268165, -1.215682, -2.670146, -0.826561, 1.570796, 1.838962],accel_mss,speed_ms,0,blend_radius_m)
    movel([0.268510, -1.212727, -2.671599, -0.828063, 1.570796, 1.839307],accel_mss,speed_ms,0,blend_radius_m)
    movel([0.269312, -1.208863, -2.673483, -0.830043, 1.570796, 1.840109],accel_mss,speed_ms,0,blend_radius_m)
    movel([0.270551, -1.205077, -2.675313, -0.831998, 1.570796, 1.841347],accel_mss,speed_ms,0,blend_radius_m)
    movel([0.272166, -1.201531, -2.677013, -0.833845, 1.570796, 1.842962],accel_mss,speed_ms,0,blend_radius_m)
    movel([0.273066, -1.199947, -2.677768, -0.834674, 1.570796, 1.843863],accel_mss,speed_ms,0,blend_radius_m)
    movel([0.274103, -1.198381, -2.678512, -0.835497, 1.570796, 1.844900],accel_mss,speed_ms,0,blend_radius_m)
    movel([0.275647, -1.196414, -2.679442, -0.836533, 1.570796, 1.846443],accel_mss,speed_ms,0,blend_radius_m)
    movel([0.277625, -1.194250, -2.680460, -0.837679, 1.570796, 1.848421],accel_mss,speed_ms,0,blend_radius_m)
    movel([0.279732, -1.192197, -2.681422, -0.838771, 1.570796, 1.850529],accel_mss,speed_ms,0,blend_radius_m)
    movel([0.281670, -1.190580, -2.682175, -0.839633, 1.570796, 1.852466],accel_mss,speed_ms,0,blend_radius_m)
    movel([0.283687, -1.189141, -2.682844, -0.840404, 1.570796, 1.854484],accel_mss,speed_ms,0,blend_radius_m)
    movel([0.285751, -1.187861, -2.683437, -0.841091, 1.570796, 1.856547],accel_mss,speed_ms,0,blend_radius_m)
    movel([0.287875, -1.186725, -2.683962, -0.841702, 1.570796, 1.858671],accel_mss,speed_ms,0,blend_radius_m)
    movel([0.290006, -1.185763, -2.684405, -0.842221, 1.570796, 1.860802],accel_mss,speed_ms,0,blend_radius_m)
    movel([0.292162, -1.184969, -2.684770, -0.842650, 1.570796, 1.862959],accel_mss,speed_ms,0,blend_radius_m)
    movel([0.294283, -1.184372, -2.685044, -0.842973, 1.570796, 1.865079],accel_mss,speed_ms,0,blend_radius_m)
    movel([0.296396, -1.183955, -2.685235, -0.843198, 1.570796, 1.867192],accel_mss,speed_ms,0,blend_radius_m)
    movel([0.298436, -1.183735, -2.685336, -0.843318, 1.570796, 1.869233],accel_mss,speed_ms,0,blend_radius_m)
    movel([0.301164, -1.183724, -2.685341, -0.843324, 1.570796, 1.871961],accel_mss,speed_ms,0,blend_radius_m)
    movel([0.303716, -1.184044, -2.685195, -0.843150, 1.570796, 1.874512],accel_mss,speed_ms,0,blend_radius_m)
    movel([0.305964, -1.184677, -2.684904, -0.842808, 1.570796, 1.876761],accel_mss,speed_ms,0,blend_radius_m)
    movel([0.307966, -1.185647, -2.684459, -0.842284, 1.570796, 1.878762],accel_mss,speed_ms,0,blend_radius_m)
    movel([0.309607, -1.186887, -2.683887, -0.841615, 1.570796, 1.880403],accel_mss,speed_ms,0,blend_radius_m)
    movel([0.310946, -1.188428, -2.683175, -0.840786, 1.570796, 1.881742],accel_mss,speed_ms,0,blend_radius_m)
    movel([0.311905, -1.190185, -2.682359, -0.839844, 1.570796, 1.882701],accel_mss,speed_ms,0,blend_radius_m)
    movel([0.312501, -1.192206, -2.681417, -0.838766, 1.570796, 1.883297],accel_mss,speed_ms,0,blend_radius_m)
    movel([0.312796, -1.195034, -2.680092, -0.837263, 1.570796, 1.883592],accel_mss,speed_ms,0,blend_radius_m)
    movel([0.312643, -1.198070, -2.678659, -0.835660, 1.570796, 1.883439],accel_mss,speed_ms,0,blend_radius_m)
    movel([0.312002, -1.202419, -2.676589, -0.833381, 1.570796, 1.882798],accel_mss,speed_ms,0,blend_radius_m)
